(* CODESYS project l2sivacuum.library
   Company: SLAC
   Title: L2SI Vacuum Library
   Placeholder: L2SI Vacuum Library
   Version: 0.0.1

Project tree, tasks and I/O mapping:
  libraries: LCLS General, 0.1.4 (SLAC); Tc2_EtherCAT, * (Beckhoff Automation GmbH); Tc2_Standard, * (Beckhoff Automation GmbH); Tc2_System, * (Beckhoff Automation GmbH); Tc2_TcpIp, * (Beckhoff Automation GmbH); Tc2_Utilities, * (Beckhoff Automation GmbH); Tc3_Interfaces, * (Beckhoff Automation GmbH); Tc3_Module, * (Beckhoff Automation GmbH)
  DUTs/
    Gauges/
      data type E_PressureState
      data type Gauge_Type
      data type ST_VG
    Pumps/
      data type E_PumpState
      data type ST_AgilentPTM
      data type ST_EbaraDryPump
      data type ST_EbaraPTM
      data type ST_LeyboldPTM
      data type ST_PfeifferPTM
      data type ST_PIP
      data type ST_PTM
      data type ST_RoughPump
    Valves/
      data type E_ValvePositionState
      data type E_VCN
      data type E_VGC
      data type ST_VCC
      data type ST_VCC_NO
      data type ST_VCN
      data type ST_VGC
      data type ST_VRC
  GVLs/
    global variables Constants
    global variables Global_Variables
  POUs/
    Functions/
      Gauges/
        function block FB_925 [ST]: ACT_IO
        function block FB_972 [ST]: ACT_IO
        function block FB_GCM [ST]: ACT_IO
        function block FB_MKS_937A [ST]
        function block FB_MKS_937B [ST]
        function block FB_MKS275 [ST]: IO
        function block FB_MKS317 [ST]: IO
        function block FB_MKS422 [ST]: IO
        function block FB_MKS500 [ST]: IO
        function block FB_MKS500_EP [ST]: IO
        function block FB_MKS722 [ST]: ACT_IO
        function block FB_PressureState [ST]
      Pumps/
        function block FB_EbaraDryPump [ST]: ACT_IO
        function block FB_PIP_Gamma [ST]: ACT_SetGauge, IO
        function block FB_PTM_Agilent [ST]: BackingPressureSetPoint, ErrorMessage, IO
        function block FB_PTM_Ebara [ST]: ACT_IO, BackingPressureSetPoint
        function block FB_PTM_MagDriveDigital [ST]: ACT_IO
        function block FB_PTM_Pfeiffer [ST]
        function block FB_ScrollPump [ST]: IO
        function block FB_TurboExtLogic [LD]
      Valves/
        function F_TURBO_VRC_ILK [ST]
        function F_VALVE_REL_ILK [ST]
        function F_VRC_DIODE_ILK [ST]
        function block FB_TurbVentvalve_NO [LD]
        function block FB_VCC [ST]: ACT_IO
        function block FB_VCN [ST]: ACT_IO
        function block FB_VGC [ST]: ACT_IO, ACT_ResetAlarms
        function block FB_VRC [ST]: ACT_IO, F_TURBO_VRC_ILK
        function block FB_VRC_OK_CLS [ST]
  Version/
    global variables Global_Version
  VISUs/
*)

// DUTs/Gauges/E_PressureState
TYPE E_PressureState :
(
	//Valid States (Positive)
	Valid := gc_GaugeValidState, // gc_GaugeValidState set in "Global Variable Folder: Constants"
	ValidHi	:= 1, //gc_GaugeValidState + 1,
	ValidLo	:= 2, //gc_GaugeValidState + 2,
	
	// Invalid states
	PressInvalid	:= -1, //gc_GaugeValidState - 1,
	GaugeDisconnected	:=	-2, //gc_GaugeValidState -2,
	OoR	:= -6, //gc_GaugeValidState -6,
	// Ion gauges
	Off		:= -3, //gc_GaugeValidState - 3,
	Starting	:= -4 //gc_GaugeValidState - 4
) INT;
END_TYPE

// DUTs/Gauges/Gauge_Type
TYPE Gauge_Type: ( 
PG722B := 0, //Baraton Gauge
IG903 := 1 , //Cold Cathode
PG907 := 2 , //Pirani Gauge
IG909:= 3 , //Hot Cathode
PG925 := 4 ); //MicroPirani Gauge
(* This enumeration should match up with the EDM MUX button on the vacuum gauge expert controls screen *)
END_TYPE

// DUTs/Gauges/ST_VG
TYPE ST_VG :
STRUCT
	/// A general gauge structure is used to make the rest of the interlocking simpler. There are some parameters for cold cathodes that are not used by pirani.
	///These features aren't disabled, they just aren't used, think child/parent classes. 
	/// 
	{attribute 'pytmc' := '
    pv: PRESS
	io: i
    '}
	rPRESS: REAL;  //This is the human-readable pressure
	{attribute 'pytmc' := '
    pv: AT_VAC
	io: i
    '}
	xAT_VAC: BOOL;
	{attribute 'pytmc' := '
    pv: PRESS_OK
	io: i
    '}
	xPRESS_OK: BOOL;
	{attribute 'pytmc' := '
    pv: STATE
	io: i
    '}
	eState	:	E_PressureState;
	(* EPICS Controls *)	
	{attribute 'pytmc' := '
    pv: HV_SW
	io: io
    '}
	xHV_SW: BOOL; // High Voltage Switch from epics
	
	/// Controls and I/Os
	{attribute 'pytmc' := '
    pv: PRESS
	io: i
    '}
	i_iPRESS_R  :INT; // input Pressure // Link to analog Input
	{attribute 'pytmc' := '
    pv: HV_ON
	io: i
    '}
	i_xHV_ON	: BOOL; //  True when High Voltage is on  // 'TcLinkTo' (EL1124) ^Input
	{attribute 'pytmc' := '
    pv: DISC_ACTIVE
	io: i
    '}
	i_xDisc_Active : BOOL;// Discharge Current Active // 'TcLinkTo' (EL1124) ^Input
	{attribute 'pytmc' := '
    pv: HV_DIS
	io: i
    '}
	q_xHV_DIS : BOOL; // Enable High Voltage when True // 'TcLinkTo' (EL2624) ^Output
	//
	wHV_RO: WORD;
		
	/// Bakeout bit 
	xBAKEOUT: BOOL;
	
	//enum for gauge type - will replace iType
	eTYPE: Gauge_Type := PG907; 
	//Gauge type, deprecated (default to pirani)
	iTYPE: INT := 2;
	// Index location of the associated Pirani Gauge
	wPG: WORD;
	
	 
	xTurnOnTime: BOOL;/// Turn on Timers for cold cathode warmup
	iVacSp	:	INT;/// At vacuum setpoint for all gauges
	{attribute 'pytmc' := '
    pv: VAC_SP
	io:io
    '}
	rVAC_SP: REAL := 0.5;
	/// Protection setpoint for ion gauges at which the gauge turns off, not used for pirani 
	{attribute 'pytmc' := '
    pv: PRO_SP
	io: io
    '}
	rPRO_SP: REAL := 0.01;
	{attribute 'pytmc' := '
    pv: SP_HYS
	io: io
    '}
	/// Protection setpoint hysteresis 
	rHYS_PR: REAL; 
	/// Full scale pressure in Torr for baratron pressure conversion 
	rFULL_SCALE: REAL := 1000;
	
END_STRUCT
END_TYPE

// DUTs/Pumps/E_PumpState
TYPE E_PumpState :
(
pumpSTOPPED	:= 0,
pumpSTARTING	:= 1,
pumpRUNNING	:= 2,
pumpFAULT := 3

);
END_TYPE

// DUTs/Pumps/ST_AgilentPTM
TYPE ST_AgilentPTM EXTENDS ST_PTM :
STRUCT

(* Inputs *)
	(* 24V in Ramp state; 0V for others *)
	{attribute 'pytmc' := '
    pv: START
	io: i
	'}
    i_xSTART :	BOOL; 
	
	(* setpoint related to frequency *)
	{attribute 'pytmc' := '
    pv: R1Status
	io: i
	'}
	i_xR1	:  BOOL;
	
	(* setpoint related to Power *)
	{attribute 'pytmc' := '
    pv: R2Status
	io: i
	'}
	i_xR2	:  BOOL;
	
	(* low speed mode *)
	{attribute 'pytmc' := '
    pv: LSPD
	io: i
	'}
	i_xLSpd	:  BOOL;
	
	{attribute 'pytmc' := '
    pv: PUMP_CURRENT
	io: i
	'}
	i_iPumpCurrent: INT;
	(* Fault input*)
	//i_xFault : BOOL;  Inherit ST_PTM.xFault
	
	

(* controls *)
	(* Start/Stop - 
		q_RunDo ;   Inherit ST_PTM.
	 *)
	
	(* Low speed control *)
	{attribute 'pytmc' := '
    pv: LSPD_DO
	io: i
	'}
	q_xLSpd		:  BOOL; 
	
	(*Soft start *)
	{attribute 'pytmc' := '
    pv: XSS_DO
	io: i
	'}
	q_xSS   	:  BOOL; 
	
	(* Run interlock*)
	{attribute 'pytmc' := '
    pv: ILK_STATUS
	io: i
	'}
	xIlk : BOOL;
	
	{attribute 'pytmc' := '
    pv: STATE
	io: i
	'}	
	eState	:	E_PumpState;
	
	
	(*pump Lock*)
	{attribute 'pytmc' := '
    pv: FaultLock
	io: i
	'}
	xPumpFaultLock : BOOL := FALSE;
	// i_xPumpLockReset: BOOL := FALSE; Inherit ST_PTM.xReset
	// Error messages
	{attribute 'pytmc' := '
    pv: ErrorMessage
	io: i
	'}
	sError : STRING;

END_STRUCT
END_TYPE

// DUTs/Pumps/ST_EbaraDryPump
TYPE ST_EbaraDryPump EXTENDS ST_RoughPump :
STRUCT
(* Extension of the rough pump archetype for ebara 
Applicable to: 
EV-S20
EV-S50
EV-S100
EV-S200
*)

//Controls
{attribute 'pytmc' := '
    pv: MPStart
	io: i
    '}
q_xMPStart	:	BOOL; //Main Pump start
{attribute 'pytmc' := '
    pv: BPStart
	io: i
    '}
q_xBPStart	:	BOOL; // Booster Pump start (this can be started by the pump automatically)

xBPIlk	:	BOOL;	//Booster pump interlock
rBPIlkSP	:	REAL := 30; //Booster pump pressure setpoint
tonBP	:	TON := (PT:=T#5S); //Timer for pressure and valve stability


//Readbacks
{attribute 'pytmc' := '
    pv: MPStatus
	io: i
    '}
i_xMPStatus	:	BOOL; //MP status
{attribute 'pytmc' := '
    pv: BPStatus
	io: i
    '}
i_xBPStatus	:	BOOL; //BP status
{attribute 'pytmc' := '
    pv: WARN
	io: i
    '}
i_xWarning	:	BOOL; //Warning status
{attribute 'pytmc' := '
    pv: ALARM
	io: i
    '}
i_xAlarm	:	BOOL; //Alarm, maps to error
{attribute 'pytmc' := '
    pv: Remote
	io: i
    '}
i_xRemote	:	BOOL; //Remote control status


END_STRUCT
END_TYPE

// DUTs/Pumps/ST_EbaraPTM
TYPE ST_EbaraPTM EXTENDS ST_PTM :
STRUCT
(* Extension of the PTM archetype for Ebara turbo controllers 
Applicable to: 
ETC series
*)
//Controls
	{attribute 'pytmc' := '
    pv: START_SW
	io: io
	'}
i_xStart   : BOOL; //Momentary start switch
	{attribute 'pytmc' := '
    pv: STOP_SW
	io: io
	'}
i_xStop    : BOOL; //Momentary stop switch
// i_xReset is momentary reset switch - resets protection functions

	{attribute 'pytmc' := '
    pv: START
	io: i
	'}
q_xStart   : BOOL; //Outputs - FB decides if these are actually set
	{attribute 'pytmc' := '
    pv: STOP
	io: i
	'}
q_xStop    : BOOL;
	{attribute 'pytmc' := '
    pv: RESET
	io: i
	'}
q_xReset   : BOOL;
	{attribute 'pytmc' := '
    pv: ILK
	io: i
	'}
q_xProtection : BOOL; //NC. If opened, pump will decelerate/not start

iq_xSpeedSet    : BOOL; //Request to set speed
q_iSpeedSet   : DINT; //Requested speed (min. 100 RPM)

i_xOverride   : BOOL; //Override mode - ignores interlocks

//Readbacks - also has Accel/At speed/Decel/Fault/Cur Speed (min 100RPM)
	{attribute 'pytmc' := '
    pv: ROTATE_STATUS
	io: i
	'}
i_xRotate : BOOL; //If open, pump is rotating
	{attribute 'pytmc' := '
    pv: DECEL
	io: i
	'}
i_xDecel  : BOOL; //If closed, brake engaged (pump decelerating)
	{attribute 'pytmc' := '
    pv: FAULT_OK
	io: i
	'}
i_xNCFault  : BOOL; //Normally closed fault wiring. If false, there is a fault, or cable is unplugged.
	{attribute 'pytmc' := '
    pv: SPEED
	io: i
	'}
i_iRawSpeed	:	INT; //Raw pump speed from analog input

END_STRUCT
END_TYPE

// DUTs/Pumps/ST_LeyboldPTM
TYPE ST_LeyboldPTM EXTENDS ST_PTM :
STRUCT
(* Extension of the PTM archetype for Oerlikon turbo controllers 
Applicable to: 
Mag Drive Digital
Mag Drive S
More?
*)
//Readbacks
	{attribute 'pytmc' := '
    pv: DECEL
	io: i
	'}
	i_xDecel	:	BOOL;
	{attribute 'pytmc' := '
    pv: TEMP
	io: i
	'}
	i_diPumpTemp:	DINT;
	{attribute 'pytmc' := '
    pv: PWR
	io: i
	'}
	i_diPwr   	:   DINT;
	i_diElecTemp:	DINT;
	{attribute 'pytmc' := '
    pv: OVR_TEMP
	io: i
	'}
	i_xTempFault:	BOOL;
	i_xNCError	:	BOOL; //Using normally closed wiring

//Controls
	{attribute 'pytmc' := '
    pv: Remote_EN
	io: io
	'}
	q_xRemote : BOOL; (* Remote control enabled *)
END_STRUCT
END_TYPE

// DUTs/Pumps/ST_PfeifferPTM
TYPE ST_PfeifferPTM EXTENDS ST_PTM :
STRUCT
(* Extension of the PTM archetype for Pfeiffer turbos 
Applicable to: 
HiPace series w/ onboard controllers
More?
*)
//Readbacks
	i_diPwr		:	DINT;
	i_diElecTemp	:	DINT;
	i_diBtmTemp:	DINT;
	i_diBrngTemp:	DINT;
	i_diMtrTemp:	DINT;
	i_iErrorCode	:	INT; //might change these to enumeration someday
	i_iWarningCode	:	INT;
	i_xTempFault	:	BOOL;
	i_uiPowerPctRbk :   UINT;
	
//Controls
	q_uiPowerPct : UINT := 100; //Should normally be 100
	
END_STRUCT
END_TYPE

// DUTs/Pumps/ST_PIP
TYPE ST_PIP :
STRUCT
(* Read back *)
// 	i_xHVisON : BOOL; 
	
(* Interlock *)
	{attribute 'pytmc' := '
    pv: ExtIlk
	io: i
	'}
   	xHV_ExtIlk : BOOL; 
	{attribute 'pytmc' := '
    pv: ENB_SP
	io: io
	'}
	rHVEna_SP : REAL := 1.0E-4;	
	
(* EPICS Controls *)	
	{attribute 'pytmc' := '
    pv: HV_SW
	io: io
    '}
	xHVEna_SW : BOOL; 
	
(* IO Controls *)
	{attribute 'pytmc' := '
    pv: HV_DO
	io: i
    '}
	q_xHVEna_DO : BOOL;	// Enable High Voltage when True // 'TcLinkTo' (EL1124) ^Input
	{attribute 'pytmc' := '
    pv: PRESS
	io: i
    '}
	i_iPRESS: REAL;  //
	{attribute 'pytmc' := '
    pv: SP_DI
	io:i
    '}
	i_xSP_DI : BOOL; // NO contact // 'TcLinkTo' (EL1004) ^Input



END_STRUCT
END_TYPE

// DUTs/Pumps/ST_PTM
TYPE ST_PTM :
STRUCT
(* General PTM Structure
Each PTM might have a serial control structure, but all will have a general supervisory control structure

NOTE: This is an archetype, use an extension of this structure for a specific pump (or make one).

*)

(* Controls *)
	{attribute 'pytmc' := '
    pv: Run_SW
	io: io
	'}
	xRunSW	:	BOOL;
	{attribute 'pytmc' := '
    pv: Reset_SW
	io: io
	'}
	xReset	:	BOOL; //For resetting faults
	{attribute 'pytmc' := '
    pv: RUN_DO
	io: i
	'}
	q_RunDO 	:	BOOL;

(* Readbacks *)
{attribute 'pytmc' := '
    pv: RUN_OK
	io: i
	'}
	xExtRunOk	:	BOOL; (* also a control *)
	{attribute 'pytmc' := '
    pv: ACCEL
	io: i
	'}
	i_xAccel	:	BOOL;
	{attribute 'pytmc' := '
    pv: AT_SPD
	io: i
	'}
	i_xAtSpd	:	BOOL;
	i_diCurSpd	:	DINT;
	
	xCommTimeout	:	BOOL := TRUE;  (* Initialized true since we haven't talked to pump yet *)
(* Alarm Outputs *)
	{attribute 'pytmc' := '
    pv: FAULT
	io: i
	'}
	i_xFault		:	BOOL; //Note, for Ebara this is *false* in a fault condition!
	{attribute 'pytmc' := '
    pv: WARN
	io: i
	'}
	i_xWarn		:	BOOL; (* warning *)
	
(* IWS instructions *)
	xActive	:	BOOL; // this bit is set to add the pump to the system
	iPumpGrp 	:	INT; // all members of a pump group start at the same time
	
(* Operational Setpoints *)
	rForelineSP	:	REAL := 0.5;
	
	{attribute 'pytmc' := '
    pv: BackingPressureSP
	io: io
	'}
	rBackingPressureSP : REAL := 0.01;
	{attribute 'pytmc' := '
    pv: InletPressureSP
	io: io
	'}
	rInletPressureSP : REAL := 0.5;
	

END_STRUCT
END_TYPE

// DUTs/Pumps/ST_RoughPump
TYPE ST_RoughPump :
STRUCT
	
(* Generic roughing pump controls 

NOTE: This is an archetype, use an extension of this structure for a specific pump (or make one).

*)

//Controls
{attribute 'pytmc' := '
    pv: RUN_SW
	io: io
	'}
pv_xRunSW	:	BOOL; //epics/ software control switch
{attribute 'pytmc' := '
    pv: RUN_DO
	io: i
	'}
q_xRunDo 	:   BOOL; 

//Status and Readback
{attribute 'pytmc' := '
    pv: ILK_OK
	io: i
	'}
xIlk	:	BOOL; //Interlock bit, true means OK to run
xExtIlk	:	BOOL; //External interlock, this is where the logic goes
{attribute 'pytmc' := '
    pv: AT_SPD
	io: i
	'}
xAtSpd	:	BOOL; //Pump at speed setpoint
{attribute 'pytmc' := '
    pv: WARN
	io: i
	'}
xWrn	:	BOOL; //Pump warning
iWrn	:	BOOL; //Warning state/code
xErr	:	BOOL; //Error summary
iErr	:	BOOL; //Error state/code

END_STRUCT
END_TYPE

// DUTs/Valves/E_ValvePositionState
TYPE E_ValvePositionState :
	(
OPEN	:= 0,
CLOSED	:= 1,
MOVING	:= 2,
INVALID :=3
	);
END_TYPE

// DUTs/Valves/E_VCN
TYPE E_VCN :
	(
CloseValve	:= 0,
ControlValve	:= 1,
OpenValve	:= 2
	);
END_TYPE

// DUTs/Valves/E_VGC
TYPE E_VGC :
(

	Vented,
	AtVacuum,
	ERR_DiffPress,
	ERR_LostVac

);
END_TYPE

// DUTs/Valves/ST_VCC
TYPE ST_VCC :
STRUCT

(* Inputs *)
{attribute 'pytmc' := '
    pv: OPN_SW
	io: io
	'}
	pv_xOPN_SW	: BOOL;
	{attribute 'pytmc' := '
    pv:OVRD_OPN
	io: io
	'}
	xOvrdOpn	:	BOOL;
	{attribute 'pytmc' := '
    pv: OPN_OK
	io: i
	'}
	xOPN_OK	: BOOL;

(* Outputs *)
{attribute 'pytmc' := '
    pv: RUN_DO
	io: i
	'}
	q_xOPN_DO	: BOOL;

END_STRUCT
END_TYPE

// DUTs/Valves/ST_VCC_NO
TYPE ST_VCC_NO :
STRUCT

(* A normally open valve needs permission to close! *)
(* Inputs *)
{attribute 'pytmc' := '
    pv: CLS_SW
	io: io
	'}
	pv_xCLS_SW	: BOOL;
	{attribute 'pytmc' := '
    pv: OVRD_CLS
	io: io
	'}
	pv_xOvrdCls	:	BOOL;
	{attribute 'pytmc' := '
    pv: CLS_OK
	io: i
	'}
	xCLS_OK	: BOOL;

(* Outputs *)
{attribute 'pytmc' := '
    pv: CLS_DO
	io: i
	'}
	xCLS_DO	: BOOL;

END_STRUCT
END_TYPE

// DUTs/Valves/ST_VCN
TYPE ST_VCN :
STRUCT
	(* VCN - Valve Controlled Needle
	Used for Pfeiffer EVR 116 needle valves *)
	{attribute 'pytmc' := '
    pv: POS_RDBK
	io: i
    '}
	// Inputs
	i_iPosition	:	INT; //Position readback (if it exists)
	
	// Outputs
	{attribute 'pytmc' := '
    pv: POS_CTRL
	io: io
    '}
	q_iRawPosition	:	INT; //Position control 
	//For the EVR 116 this is 0-10V analog
	
	//Softvariables
	{attribute 'pytmc' := '
    pv: ILK_OK
	io: i
    '}
	xIlk	:	BOOL := FALSE; // Interlock Bit
	rUpperLimit	:	REAL;	//Upper limit on valve open
	rReqPosition	:	REAL; //Requested position (0.0-100.0%)
	eValveControl	:	E_VCN := CloseValve; // Valve control state

	ftIlk	:	F_TRIG;	

END_STRUCT
END_TYPE

// DUTs/Valves/ST_VGC
TYPE ST_VGC :
STRUCT

(* I/Os*)
(* Readbacks *)
	{attribute 'pytmc' := '
    pv: OPN_DI
	io: i
    '}
	i_xOpnLS	: BOOL;
	{attribute 'pytmc' := '
    pv: CLS_DI
	io: i
    '}
	i_xClsLS	: BOOL;
(* Controls *)
	{attribute 'pytmc' := '
    pv: OPN_DO
	io: i
    '}
	q_xOPN_DO	: BOOL;
	
	
(* EPICS Controls *)
	{attribute 'pytmc' := '
    pv: OPN_SW
	io: o
    '}
	pv_xOPN_SW	: BOOL;
	{attribute 'pytmc' := '
    pv: ALM_RST
	io: o
    '}
	pv_xAlmRst	: BOOL;
	{attribute 'pytmc' := '
    pv: OVRD_OPN
	io: o
    '}
	pv_xOvrdOpn	:	BOOL;

(* Interlocks *)
	{attribute 'pytmc' := '
    pv: DP_OK
	io: i
    '}
	xDP_OK	:	BOOL;	(* Managed by the VGC function (FB_VGC) *)// Indicates the valve can be opened because the differential pressure is low enough
	xEXT_OK	:	BOOL := FALSE;	(* External interlock for custom interlocking in addition to regular DP ilk, this must be set true, or the interlock condition before calling the FB_VGC *)
	{attribute 'pytmc' := '
    pv: OPN_OK
	io: i
    '}
	xOPN_OK	:	BOOL;	(* Final SUM of DP_OK and EXT_OK, needed because it allows the DP ilk to be switched off, see FB_VGC.Dis_DPIlk *)
	{attribute 'pytmc' := '
    pv: AT_VAC_SP
	io: o
    '}
	rAT_VAC_SP	:	REAL := 0.01;	// Interlock setpoint for gauges on both sides of valve
	rAT_VAC_SP_LAST	:	REAL :=0.01 ;	// Interlock setpoint for gauges on both sides of valve
	{attribute 'pytmc' := '
    pv: AT_VAC_HYS
	io: o
    '}
	rAT_VAC_HYS	:	REAL :=0.01;	// Hysteresis of the vacuum sp
	{attribute 'pytmc' := '
    pv: HYST_PERC
	io: o
    '}
	rHYST_PERC	:	REAL := 0.80;	// Hysteresis percentage
	{attribute 'pytmc' := '
    pv: AT_VAC
	io: i
    '}
	xAT_VAC	:	BOOL;	//At vacuum setpoint


(* Alarm Outputs *)
	xERR_DifPres		: 	BOOL;
	xERR_LstVac		: 	BOOL;
	xAlmSum			: 	BOOL;
	

	bErrorPresent : BOOL;
	iErrorCode: INT;
	sErrorMessage: STRING;

(*State*)	
	{attribute 'pytmc' := '
    pv: STATE
	io: i
    '}
	eVGC_State : E_VGC;
	{attribute 'pytmc' := '
    pv: POS_STATE
	io: i
    '}
	eState	:	E_ValvePositionState := INVALID;
	
END_STRUCT
END_TYPE

// DUTs/Valves/ST_VRC
TYPE ST_VRC :
STRUCT
(* Readbacks *)
	//If True, Valve is Open
	{attribute 'pytmc' := '
    pv: OPN_DI
	io: i
    '}
	i_xOpnLS	:	BOOL;
	//If True, Valve is Closed
	{attribute 'pytmc' := '
    pv: CLS_DI
	io: i
    '}
	i_xClsLS	:	BOOL;
	
	{attribute 'pytmc' := '
    pv: POS_STATE
	io: i
    '}
	eState	:	E_ValvePositionState := INVALID;

(* Inputs *)
	//Manually Pressing valve "Open/Close" on EDM
	{attribute 'pytmc' := '
    pv: OPN_SW
	io: io
    '}
	pv_xOPN_SW	: BOOL;
	//Manually toggling valve Local "ILK on button" on EDM
	{attribute 'pytmc' := '
    pv: OVRD_OPN
	io: io
    '}
	pv_xOvrdOpn	:	BOOL;
	//Calculated permissions to open valve
	{attribute 'pytmc' := '
    pv: OPN_OK
	io: i
    '}
	xOPN_OK	: BOOL;
	//In case VRC is normally open
	{attribute 'pytmc' := '
    pv: CLS_OK
	io: i
    '}
	xCLS_OK : BOOL := TRUE;
(* Outputs *)
	//When True, Opens valve
	//When False, Closes valve
	{attribute 'pytmc' := '
    pv: OPN_DO
	io: i
    '}
	q_xOPN_DO	: BOOL;

END_STRUCT
END_TYPE

// GVLs/Constants
VAR_GLOBAL CONSTANT
	gc_iSizeOfGGOArray : INT := 50;
	gc_GaugeValidState :	INT := 0;
END_VAR

// GVLs/Global_Variables
VAR_GLOBAL
	g_iSizeOfGGOArray : INT := 50;
	
	g_stSystem	:	System_Struct:= (
    	xFirstScan := TRUE
	);
	
	g_DummyVG	:	ST_VG;
	
	
	 fbGetCurTaskIdx : GETCURTASKINDEX;

END_VAR

// Version/Global_Version
{attribute 'TcGenerated'}
// This function has been automatically generated from the project information.
VAR_GLOBAL CONSTANT
	{attribute 'const_non_replaced'}
	{attribute 'linkalways'}
	stLibVersion_L2SI_Vacuum_Library : ST_LibVersion := (iMajor := 0, iMinor := 0, iBuild := 1, iRevision := 0, sVersion := '0.0.1');
END_VAR

// POUs/Functions/Gauges/FB_925
FUNCTION_BLOCK FB_925
VAR_INPUT
END_VAR
VAR_OUTPUT
	{attribute 'pytmc' := '
    pv: 
	'}
	PG	: ST_VG;
END_VAR
VAR_IN_OUT
	
END_VAR
VAR
	rV : REAL;
	fbGaugeState : FB_PressureState;
	rMaxPressure	:	REAL := 760; //Torr
	rMinPressure	:	REAL := 1E-5; //Torr
	
	(*IO*)
	i_iPRESS_R AT%I* :INT; // input Pressure // Link to analog Input
END_VAR

(* Standard MKS 9XX series conversion *)
(* works for 972 and 925 *)

//Default setpoint 50 mT
IF PG.rVAC_SP = 0 THEN
	PG.rVAC_SP := 5E-2;
END_IF

rV := 10*INT_TO_REAL(PG.i_iPRESS_R)/32767;

IF rV >= 0.99 THEN
	IF rV >= 0.99 AND rV < 1 THEN
		PG.rPRESS := 1E-5;
	ELSE
		PG.rPRESS := LREAL_TO_REAL(EXPT(10, rV-6));
	END_IF
	PG.xPRESS_OK := TRUE; //Backwards compatibility
ELSE
	PG.xPRESS_OK := FALSE;
END_IF

(* Pressure OK check *)
fbGaugeState.i_rV := rV;
fbGaugeState.i_MaxPressure := rMaxPressure;
fbGaugeState.i_MinPressure := rMinPressure;
fbGaugeState(iq_stVG:=PG);

(* Setpoint evaluation *)
PG.xAT_VAC := PG.xPRESS_OK AND (PG.rPRESS < PG.rVAC_SP);

ACTION ACT_IO:
PG.i_iPRESS_R :=i_iPRESS_R;
END_ACTION

END_FUNCTION_BLOCK

// POUs/Functions/Gauges/FB_PressureState
FUNCTION_BLOCK FB_PressureState
VAR_INPUT
	i_rV	:	REAL;
	i_rVMin	:	REAL := 0.01; // Anything less than this voltage is considered disconnected
	i_rVMax :	REAL := 10.5; // Anything more than this is considered invalid
	i_IGTurnOnTime	:	TIME := T#10S;
	
	i_MinPressure	:	REAL;
	i_MaxPressure	:	REAL;
END_VAR
VAR_OUTPUT
	q_eState 	:	E_PressureState;
END_VAR
VAR_IN_OUT
	iq_stVG	:	ST_VG;
END_VAR
VAR
	tonGaugeTurnOnTmr : TON;
END_VAR

(* Pressure State Evaluation
A. Wallace, 2016-8-31

This FB serves to evaluate the state of the pressure based on the raw voltage, pressure, and gauge state.

*)
// Is the gauge plugged in, and within a reasonable range?
IF i_rV < i_rVMin THEN
	q_eState := GaugeDisconnected;
ELSIF i_rV > i_rVMax THEN
	q_eState := PressInvalid;
ELSE
	// Is the gauge reading back a pressure that makes sense?
	CASE iq_stVG.eTYPE OF
		IG903:
			tonGaugeTurnOnTmr(IN:=iq_stVG.q_xHV_DIS, PT:=i_IGTurnOnTime, Q=>iq_stVG.xTurnOnTime);
			IF iq_stVG.q_xHV_DIS THEN
				IF tonGaugeTurnOnTmr.Q THEN
					IF iq_stVG.rPRESS >= i_MinPressure AND iq_stVG.rPRESS <= i_MaxPressure THEN
						q_eState := Valid;
					ELSE
						q_eState := OoR; 
					END_IF
				ELSE
						q_eState := Starting;
				END_IF
			ELSE
				q_eState := Off;
			END_IF
		IG909:
			IF iq_stVG.q_xHV_DIS THEN
				IF iq_stVG.rPRESS >= i_MinPressure AND iq_stVG.rPRESS <= i_MaxPressure THEN
					q_eState := Valid;
				ELSE
					q_eState := OoR;
				END_IF
			ELSE
				q_eState := Off;
			END_IF
		PG907, PG925, PG722B:
			IF iq_stVG.rPRESS >= i_MinPressure AND iq_stVG.rPRESS <= i_MaxPressure THEN
				q_eState := Valid;
			ELSIF iq_stVG.rPRESS < i_MinPressure THEN
				q_eState := ValidLo;
			ELSE
				q_eState := ValidHi;
			END_IF
		ELSE
			q_eState := PressInvalid;
	END_CASE
END_IF


iq_stVG.eState := q_eState;

// Legacy Press OK boolean eval
iq_stVG.xPRESS_OK := q_eState >= gc_GaugeValidState;

END_FUNCTION_BLOCK

// POUs/Functions/Gauges/FB_972
FUNCTION_BLOCK FB_972
VAR_INPUT
END_VAR
VAR_OUTPUT
	{attribute 'pytmc' := '
    pv: 
	'}
	VG	: ST_VG;
END_VAR
VAR_IN_OUT
	
END_VAR
VAR
	rV : REAL;
	(*IO*)
	i_iPRESS_R AT%I* :INT; // input Pressure // Link to analog Input
END_VAR

(* Standard MKS 9XX series conversion *)
(* works for 972 and 925 *)

rV := 10*INT_TO_REAL(VG.i_iPRESS_R)/32767;

IF rV > 1 THEN
	VG.rPRESS := LREAL_TO_REAL(EXPT(10, 2*rV-11));
	VG.xPRESS_OK := TRUE;
	VG.eState := Valid; //Press OK
ELSE
	VG.xPRESS_OK := FALSE;
	VG.eState := -6;
END_IF

ACTION ACT_IO:
VG.i_iPRESS_R :=i_iPRESS_R;
END_ACTION

END_FUNCTION_BLOCK

// POUs/Functions/Gauges/FB_GCM
FUNCTION_BLOCK FB_GCM
VAR_IN_OUT

END_VAR
VAR_OUTPUT
		{attribute 'pytmc' := '
    pv: 
	'}
	VG	:	ST_VG;
END_VAR
VAR
	rMinPressure: REAL;
	rV	:REAL;
	
	(*IO*)
	i_iPRESS_R AT%I* :INT; // input Pressure // Link to analog Input
END_VAR

(* Baratron Pressure Calc 
A. Wallace
2016-6-16
The full-scale pressure times the ratio of the meas.
voltage to full-scale voltage (10V).
The minimum pressure is always going to be 5e-4 * F.S.V.*)

rMinPressure := VG.rFULL_SCALE * 5E-4;


rV :=MAX((10*INT_TO_REAL(VG.i_iPRESS_R)/32767),0);
VG.rPRESS := (VG.rFULL_SCALE/10)*rV;
IF VG.rPRESS > rMinPressure THEN
	VG.xPRESS_OK := TRUE;
ELSE
	VG.xPRESS_OK := FALSE;
END_IF

(*IO soft linking*)
ACT_IO();

ACTION ACT_IO:
VG.i_iPRESS_R :=i_iPRESS_R;
END_ACTION

END_FUNCTION_BLOCK

// POUs/Functions/Gauges/FB_MKS_937A
FUNCTION_BLOCK FB_MKS_937A
VAR_IN_OUT
	VG : ST_VG;
END_VAR
VAR_INPUT
	PG	:	ST_VG := g_DummyVG;
END_VAR
VAR_OUTPUT
END_VAR
VAR
	rV	:	REAL;
END_VAR

(* 937A Logarithmic Output Conversion *)
(* 7-15-2015 *)
(* This function will read the pressure from any gauge on a 937A. *)

rV := 10*INT_TO_REAL(VG.i_iPRESS_R)/32767;
VG.rPRESS := LREAL_TO_REAL(EXPT(10,rV/0.6-12));


(* Ion Gauge Protection Functions *)
(* If the PG pressure is greater than the VG.PRO_SP then the gauge is disabled *)
(* If the PG pressure is less than the VG.PRO_SP then the gauge is enabled *)
(* This FB also implements some hysteresis so the gauge doesn't have rapid power cycling while near the turn on boundary *)

IF PG.rPRESS < VG.rPRO_SP THEN

VG.q_xHV_DIS := NOT VG.xHV_SW;

ELSIF NOT VG.q_xHV_DIS THEN
	IF VG.rPRESS > VG.rPRO_SP + VG.rHYS_PR OR PG.rPRESS > VG.rPRO_SP + VG.rHYS_PR THEN
		VG.q_xHV_DIS := TRUE;
	END_IF
ELSE
	VG.q_xHV_DIS := TRUE;
END_IF


(* Pressure gauge OK checks *)
VG.xPRESS_OK := (rV <=9.6 ) AND (rV>=0.6); //legacy

IF (rV <=9.6 ) AND (rV>=0.6) THEN
	VG.eState := Valid; // normal
ELSIF rV >= 0.18 AND rV <= 0.22 THEN
	VG.eState := ValidLo; //LO
ELSIF rV >= 9.7 AND rV<= 9.9 THEN
	VG.eState := ValidHi; //HIGH
ELSIF rV < 0.18 THEN
	VG.eState := GaugeDisconnected; //not on
ELSE
	VG.eState := PressInvalid; //other fault - could be no gauge, controller powering up etc
END_IF

(* Setpoint evaluation *)
VG.xAT_VAC := (VG.eState =Valid) AND VG.rPRESS < VG.rVAC_SP;

END_FUNCTION_BLOCK

// POUs/Functions/Gauges/FB_MKS_937B
FUNCTION_BLOCK FB_MKS_937B
VAR_IN_OUT
	
		PG	:	ST_VG := g_DummyVG;
END_VAR
VAR_INPUT
	
END_VAR
VAR_OUTPUT
	{attribute 'pytmc' := '
    pv: GCC
	'}
	VG : ST_VG;
	
	

END_VAR
VAR
	rV	:	REAL;
END_VAR

(* 937B Logarithmic Output Conversion *)
(* 5-20-2016, Alex Wallace and Scott Stubbs *)
(* This function will read the pressure from any gauge on a 937B. *)

rV := 10*INT_TO_REAL(VG.i_iPRESS_R)/32767;
VG.rPRESS := LREAL_TO_REAL(EXPT(10,(rV-7.2)/0.6));


(* Ion Gauge Protection Functions *)
(* If the PG pressure is greater than the VG.PRO_SP then the gauge is disabled *)
(* If the PG pressure is less than the VG.PRO_SP then the gauge is enabled *)
(* This FB also implements some hysteresis so the gauge doesn't have rapid power cycling while near the turn on boundary *)

IF PG.rPRESS < VG.rPRO_SP THEN

VG.q_xHV_DIS := NOT VG.xHV_SW;

ELSIF NOT VG.q_xHV_DIS THEN
	IF VG.rPRESS > VG.rPRO_SP + VG.rHYS_PR OR PG.rPRESS > VG.rPRO_SP + VG.rHYS_PR THEN
		VG.q_xHV_DIS := TRUE;
	END_IF
ELSE
	VG.q_xHV_DIS := TRUE;
END_IF


(* Pressure gauge OK checks *)
VG.xPRESS_OK := (rV <=9.6 ) AND (rV>=0.6);

IF (rV <=9.7 ) AND (rV>=0.6) THEN
	VG.eState := Valid; // normal
ELSIF rV >= 0.18 AND rV <= 0.22 THEN
	VG.eState := ValidLo; //LO
ELSIF rV > 9.7 AND rV<= 9.9 THEN
	VG.eState := ValidHi; //HIGH
ELSIF rV < 0.18 THEN
	VG.eState := GaugeDisconnected; //not on
ELSE
	VG.eState := PressInvalid; //other fault - could be no gauge, controller powering up etc
END_IF

(* Setpoint evaluation *)
VG.xAT_VAC := (VG.eState =Valid) AND VG.rPRESS < VG.rVAC_SP;

END_FUNCTION_BLOCK

// POUs/Functions/Gauges/FB_MKS275
FUNCTION_BLOCK FB_MKS275
VAR_IN_OUT

END_VAR
VAR_INPUT
END_VAR

VAR_OUTPUT
	{attribute 'pytmc' := '
    pv: 
	'}
	PG : ST_VG;
END_VAR
VAR
	MinPressure: REAL := 1E-4;
	V : REAL;
	Vlowest: REAL := 10;
	
	rValidLoBoundary	:	REAL := 0.375; // manual page 27
	rValidHiBoundary	:	REAL := 5.659;// 5.534; // manual page 27
	rDisconnectedBoundary	:	REAL := 0.3;
	
	(*IO*)
	i_iPRESS_R AT%I* :INT; // input Pressure // Link to analog Input
END_VAR

(* This function block is used to provide protection and automatic turn on of ion gauges,
 it also manages the turn on of the AT_VAC boolean, and checks to make sure the pressure is good *)
(* For MKS 275 mini-convectron *)

//Default setpoint 50 mT
IF PG.rVAC_SP = 0 THEN
	PG.rVAC_SP := 5E-2;
END_IF

(* Real-value calculation *)

V := 10*INT_TO_REAL(PG.i_iPRESS_R)/32767;	

Vlowest := MIN(V, Vlowest);

IF V > rDisconnectedBoundary AND V < rValidLoBoundary THEN

PG.rPRESS := MinPressure;
PG.eState := ValidLo;

ELSIF V >= rValidLoBoundary AND V < 2.842 THEN

PG.rPRESS := MAX( MinPressure, LREAL_TO_REAL( -0.02585 + 0.03767*V + 0.04563*EXPT(V,2)+ 0.1151*EXPT(V,3) - 0.04158*EXPT(V,4)+ 0.008737*EXPT(V,5)) );
PG.eState := Valid;

ELSIF V >= 2.842 AND V < 4.945 THEN

PG.rPRESS := LREAL_TO_REAL((0.1031-0.02322*V+0.07229*EXPT(V,2))/(1-0.3986*V+0.07438*EXPT(V,2)-0.006866*EXPT(V,3)));
PG.eState := Valid;

ELSIF V >= 4.945 AND V < rValidHiBoundary THEN

PG.rPRESS := LREAL_TO_REAL((100.624-20.5623*V)/(1-0.37679*V+0.0348656*EXPT(V,2)));
PG.eState := Valid;

ELSIF V <= rDisconnectedBoundary THEN

PG.eState := GaugeDisconnected; //Most likely not connected
PG.rPRESS := -1;;

ELSE
	
PG.eState := OoR; //Larger voltage, probably out of range?
PG.rPRESS := -1;
END_IF

(* Protection Functions *)
(* If the PG pressure is greater than the IG.PRO_SP then the gauge is disabled *)
(* If the PG pressure is less than the IG.PRO_SP then the gauge is enabled *)
(* This FB also implements some hysteresis so the gauge doesn't have rapid power cycling while near the turn on boundary *)

(* Pressure OK check *)
PG.xPRESS_OK := (PG.rPRESS >= MinPressure);

(* Setpoint evaluation *)
PG.xAT_VAC := PG.xPRESS_OK AND (PG.rPRESS<PG.rVAC_SP);

(*Soft IO Mapping *)
IO();

ACTION IO:
PG.i_iPRESS_R :=i_iPRESS_R;
END_ACTION

END_FUNCTION_BLOCK

// POUs/Functions/Gauges/FB_MKS317
FUNCTION_BLOCK FB_MKS317
VAR_IN_OUT
	
END_VAR
VAR_INPUT
	
END_VAR
VAR_OUTPUT
	{attribute 'pytmc' := '
    pv: 
	'}
	PG : ST_VG;
END_VAR
VAR
	rV	:	REAL;
		MinPressure: REAL := 1E-4;
		(*IO*)
	i_iPRESS_R AT%I* :INT; // input Pressure // Link to analog Input
END_VAR

(* 937B Logarithmic Output Conversion *)
(* 5-20-2016, Alex Wallace and Scott Stubbs *)
(* 09-28-2018, Margaret Ghaly *)
(* This function will read the pressure from any gauge on a 937B. *)

rV := 10*INT_TO_REAL(PG.i_iPRESS_R)/32767;
PG.rPRESS := LREAL_TO_REAL(EXPT(10,(rV-7.2)/0.6));


//Default setpoint 50 mT
IF PG.rVAC_SP = 0 THEN
	PG.rVAC_SP := 5E-2;
END_IF


(* Pressure gauge OK checks *)
PG.xPRESS_OK := (rV <=9.6 ) AND (rV>=0.6);

IF (rV <=9.7 ) AND (rV>=0.6) THEN
	PG.eState := Valid; // normal
ELSIF rV >= 0.18 AND rV <= 0.22 THEN
	PG.eState := ValidLo; //LO
ELSIF rV > 9.7 AND rV<= 9.9 THEN
	PG.eState := ValidHi; //HIGH
ELSIF rV < 0.18 THEN
	PG.eState := GaugeDisconnected; //not on
ELSE
	PG.eState := PressInvalid; //other fault - could be no gauge, controller powering up etc
END_IF

(* Pressure OK check *)
PG.xPRESS_OK := (PG.rPRESS >= MinPressure);

(* Setpoint evaluation *)
PG.xAT_VAC := (PG.eState =Valid) AND PG.rPRESS < PG.rVAC_SP;

ACTION IO:
PG.i_iPRESS_R :=i_iPRESS_R;
END_ACTION

END_FUNCTION_BLOCK

// POUs/Functions/Gauges/FB_MKS422
FUNCTION_BLOCK FB_MKS422
VAR_IN_OUT
		
END_VAR
VAR_INPUT
		PG	:	ST_VG;
END_VAR
VAR_OUTPUT
	{attribute 'pytmc' := '
    pv: GCC
	'}
	IG : ST_VG;
END_VAR
VAR
	rV	:	REAL;
	
	(*IOs to be linked*)
	/// Controls and I/Os
	i_iPRESS_R AT %I* :INT; // input Pressure // Link to analog Input
	q_xHV_DIS AT %Q* : BOOL; // Enable High Voltage when True // 'TcLinkTo' (EL2624) ^Output
	
	
END_VAR

(* 937B Logarithmic Output Conversion *)
(* 5-20-2016, Alex Wallace and Scott Stubbs *)
(* 09-28-2018, Margaret Ghaly *)
(* This function will read the pressure from any gauge on a 937B. *)

rV := 10*INT_TO_REAL(IG.i_iPRESS_R)/32767;
IG.rPRESS := LREAL_TO_REAL(EXPT(10,(rV-7.2)/0.6));



IF (rV <=9.7 ) AND (rV>=0.6) THEN
	IG.eState := Valid; // normal
ELSIF rV >= 0.18 AND rV <= 0.22 THEN
	IG.eState := ValidLo; //LO
ELSIF rV > 9.7 AND rV<= 9.9 THEN
	IG.eState := ValidHi; //HIGH
ELSIF rV < 0.18 THEN
	IG.eState := GaugeDisconnected; //not on
ELSE
	IG.eState := PressInvalid; //other fault - could be no gauge, controller powering up etc
END_IF


(* Ion Gauge Protection Functions *)
(* If the PG pressure is greater than the VG.PRO_SP then the gauge is disabled *)
(* If the PG pressure is less than the VG.PRO_SP then the gauge is enabled *)
(* This FB also implements some hysteresis so the gauge doesn't have rapid power cycling while near the turn on boundary *)

IF PG.rPRESS < IG.rPRO_SP THEN
	IG.q_xHV_DIS := IG.xHV_SW;

ELSIF IG.q_xHV_DIS THEN
	IF IG.rPRESS > (IG.rPRO_SP + IG.rHYS_PR) OR PG.rPRESS > (IG.rPRO_SP + IG.rHYS_PR) THEN
		IG.q_xHV_DIS := FALSE;
		IG.xHV_SW := FALSE;
	END_IF
ELSE
	IG.xHV_SW := FALSE;
END_IF

(* Pressure gauge OK checks *)
IG.xPRESS_OK := (rV <=9.6 ) AND (rV>=0.6);


(* Setpoint evaluation *)
IG.xAT_VAC := IG.xPRESS_OK AND IG.rPRESS < IG.rVAC_SP;


(*Soft IO Linking*)
// check ethercat Diagnostics
IO();

ACTION IO:
(*soft link inputs*)
IG.i_iPRESS_R:=	i_iPRESS_R; 

(*soft link outputs*)
q_xHV_DIS := IG.q_xHV_DIS;
END_ACTION

END_FUNCTION_BLOCK

// POUs/Functions/Gauges/FB_MKS500
FUNCTION_BLOCK FB_MKS500
VAR_IN_OUT

END_VAR
VAR_INPUT
	PG	:	ST_VG;
END_VAR
VAR_OUTPUT
	{attribute 'pytmc' := '
    pv: 
	'}
	IG : ST_VG;
END_VAR
VAR
	rV : REAL;
	pBase : REAL :=1.0E-10;//default curve base pressure is 1E-10. Confusing since can't actually read that low using analog out.
	vBase : REAL := 0; // corresponding vbase 0V based on default curve.  See manual pg. 44
	vSlope : REAL := 1.0; //looks correct for default curve
	GaugeTurnOnTmr : TON;
	MinPressure: REAL := 1E-10;
	cDefaultPressure : REAL := 0;
	
	
	(*IOs to be linked*)
	/// Controls and I/Os
	i_iPRESS_R AT %I* :INT; // input Pressure // Link to analog Input
	i_xHV_ON AT %I*	: BOOL; //  True when High Voltage is on  // 'TcLinkTo' (EL1124) ^Input
	i_xDisc_Active AT %I* : BOOL;// Discharge Current Active // 'TcLinkTo' (EL1124) ^Input
	q_xHV_DIS AT %Q* : BOOL; // Enable High Voltage when True // 'TcLinkTo' (EL2624) ^Output
	//
END_VAR

(* 500 Logarithmic Output Conversion, factory default configuration *)

rV := 10*INT_TO_REAL(IG.i_iPRESS_R)/32767;

(*
IF rV >= 0.49 AND rV < 0.52  THEN
	IG.wState := 5;
	IG.rPRESS := cDefaultPressure;
ELSIF rV < 0.4 THEN
	IG.wState := 4;//HV Off/ gauge disconnected
	IG.rPRESS := cDefaultPressure;
ELSE
	IG.wState := 1;
	IG.rPRESS := LREAL_TO_REAL(EXPT(10,((rV-vBase)/vSlope+LOG(pBase))));
END_IF
*)

(* Set Guage State based on the inputs HV ON and Discharge current*)
IF IG.i_xHV_ON AND NOT IG.i_xDisc_Active THEN
	IG.eState := Starting;
	IG.rPRESS := cDefaultPressure;
ELSIF IG.i_xHV_ON AND IG.i_xDisc_Active THEN
	IG.eState := Valid;
	IG.rPRESS := LREAL_TO_REAL(EXPT(10,((rV-vBase)/vSlope+LOG(pBase))));
ELSIF NOT IG.i_xHV_ON AND NOT IG.i_xDisc_Active THEN
	IG.eState := Off;
	IG.rPRESS := cDefaultPressure;
END_IF




(* Ion Gauge Protection Functions *)
(* If the PG pressure is greater than the VG.PRO_SP then the gauge is disabled *)
(* If the PG pressure is less than the VG.PRO_SP then the gauge is enabled *)
(* This FB also implements some hysteresis so the gauge doesn't have rapid power cycling while near the turn on boundary *)



IF PG.rPRESS < IG.rPRO_SP AND PG.xPRESS_OK THEN

	IG.q_xHV_DIS := IG.xHV_SW;

ELSIF IG.q_xHV_DIS THEN
	IF IG.rPRESS > (IG.rPRO_SP + IG.rHYS_PR)  OR PG.rPRESS > (IG.rPRO_SP + IG.rHYS_PR) THEN
		IG.q_xHV_DIS := FALSE;
		IG.xHV_SW := FALSE;
	END_IF
ELSE
	IG.q_xHV_DIS := FALSE;
	IG.xHV_SW := FALSE;
END_IF

(* Pressure gauge OK checks *)

GaugeTurnOnTmr(IN:=IG.q_xHV_DIS, PT:=T#10S, Q=>IG.xTurnOnTime);


//Backwards compatibility
IG.xPRESS_OK := (IG.eState = Valid) OR IG.xBAKEOUT;

(* Setpoint evaluation *)
IG.xAT_VAC := (IG.xPRESS_OK AND (IG.rPRESS < IG.rVAC_SP)) OR IG.xBAKEOUT AND (IG.eState = Valid) ;


(*Soft IO Linking*)
// check ethercat Diagnostics
IO();

ACTION IO:
(*check health of the ethercat terminal*) //todo
(*soft link inputs*)
IG.i_iPRESS_R:=	i_iPRESS_R; 
IG.i_xHV_ON:= i_xHV_ON;
IG.i_xDisc_Active:=i_xDisc_Active; 
(*soft link outputs*)
q_xHV_DIS := IG.q_xHV_DIS;
END_ACTION

END_FUNCTION_BLOCK

// POUs/Functions/Gauges/FB_MKS500_EP
FUNCTION_BLOCK FB_MKS500_EP
VAR_IN_OUT
		
END_VAR
VAR_INPUT

	PG	:	ST_VG;
END_VAR
VAR_OUTPUT
{attribute 'pytmc' := '
    pv: 
	'}
	IG : ST_VG;
END_VAR
VAR
	rV : REAL;
	pBase : REAL :=1.0E-10;//default curve base pressure is 1E-10. Confusing since can't actually read that low using analog out.
	vBase : REAL := 0; // corresponding vbase 0V based on default curve.  See manual pg. 44
	vSlope : REAL := 1.0; //looks correct for default curve
	GaugeTurnOnTmr : TON;
	MinPressure: REAL := 1E-10;
	cDefaultPressure : REAL := 0;
	
	
	(*IOs to be linked*)
	/// Controls and I/Os
	i_iPRESS_R AT %I* :INT; // input Pressure // Link to analog Input
	q_xHV_DIS AT %Q* : BOOL; // Enable High Voltage when True // 'TcLinkTo' (EP2624) ^Output
	//
END_VAR

(* 500 Logarithmic Output Conversion, factory default configuration *)


(*check health of the ethercat terminal*)

rV := 10*INT_TO_REAL(IG.i_iPRESS_R)/32767;

(* Set Guage State based on the inputs HV ON and Discharge current*)
IF rV >= 0.49 AND rV < 0.6  THEN
	IG.eState := Starting;
	IG.rPRESS := cDefaultPressure;
ELSIF rV < 0.4 THEN
	IG.eState := Off;
	IG.rPRESS := cDefaultPressure;
ELSE
	IG.eState := Valid;
	IG.rPRESS := LREAL_TO_REAL(EXPT(10,((rV-vBase)/vSlope+LOG(pBase))));
END_IF



(* Ion Gauge Protection Functions *)
(* If the PG pressure is greater than the VG.PRO_SP then the gauge is disabled *)
(* If the PG pressure is less than the VG.PRO_SP then the gauge is enabled *)
(* This FB also implements some hysteresis so the gauge doesn't have rapid power cycling while near the turn on boundary *)



IF PG.rPRESS < IG.rPRO_SP AND PG.xPRESS_OK THEN

	IG.q_xHV_DIS := IG.xHV_SW;

ELSIF IG.q_xHV_DIS THEN
	IF IG.rPRESS > (IG.rPRO_SP + IG.rHYS_PR)  OR PG.rPRESS > (IG.rPRO_SP + IG.rHYS_PR) THEN
		IG.q_xHV_DIS := FALSE;
		IG.xHV_SW := FALSE;
	END_IF
ELSE
	IG.q_xHV_DIS := FALSE;
	IG.xHV_SW := FALSE;
END_IF

(* Pressure gauge OK checks *)

GaugeTurnOnTmr(IN:=IG.q_xHV_DIS, PT:=T#10S, Q=>IG.xTurnOnTime);


//Backwards compatibility
IG.xPRESS_OK := (IG.eState = Valid) OR IG.xBAKEOUT;

(* Setpoint evaluation *)
IG.xAT_VAC := (IG.xPRESS_OK AND (IG.rPRESS < IG.rVAC_SP)) OR IG.xBAKEOUT AND (IG.eState = Valid) ;


(*Soft IO Linking*)
// check ethercat Diagnostics
IO();

ACTION IO:
(*soft link inputs*)
IG.i_iPRESS_R:=	i_iPRESS_R; 
(*soft link outputs*)
q_xHV_DIS := IG.q_xHV_DIS;
END_ACTION

END_FUNCTION_BLOCK

// POUs/Functions/Gauges/FB_MKS722
FUNCTION_BLOCK FB_MKS722
VAR_IN_OUT
	
END_VAR
VAR_OUTPUT
	{attribute 'pytmc' := '
    pv: 
	'}
	VG	:	ST_VG;
END_VAR
VAR_INPUT
	i_rMinPressure	:	REAL;
	i_rMaxPressure	:	REAL;
END_VAR
VAR
	rMinPressure: REAL;
	rVMin	:	REAL := 0.01; // Anything less than this voltage is considered disconnected
	rVMax :	REAL := 10.5; // Anything more than this is considered invalid
	rV	:REAL;
	
	(*IO*)
	i_iPRESS_R AT%I* :INT; // input Pressure // Link to analog Input
END_VAR


// Is the gauge plugged in, and within a reasonable range?
IF rV < rVMin THEN
	VG.eState := GaugeDisconnected;
ELSIF rV > rVMax THEN
	VG.eState := PressInvalid;
ELSIF VG.rPRESS >= rMinPressure AND VG.rPRESS <= i_rMaxPressure THEN
				VG.eState := Valid;
ELSIF VG.rPRESS < i_rMinPressure THEN
				VG.eState := ValidLo;
ELSE
				VG.eState := ValidHi;
END_IF
			
// Legacy Press OK boolean eval
VG.xPRESS_OK := VG.eState >= gc_GaugeValidState;

(*IO Soft Mapping*)
ACT_IO();

ACTION ACT_IO:
VG.i_iPRESS_R :=i_iPRESS_R;
END_ACTION

END_FUNCTION_BLOCK

// POUs/Functions/Pumps/FB_EbaraDryPump
FUNCTION_BLOCK FB_EbaraDryPump
VAR_INPUT
	i_stBPGauge	:	ST_VG; //booster pump interlock gauge
	i_xVlvOpn	:	BOOL; //valve(s) to main system load are open
END_VAR
VAR_OUTPUT
END_VAR
VAR_IN_OUT
	{attribute 'pytmc' := '
    pv: 
	'}
	stPump	:	ST_EbaraDryPump; //Ebara dry pump structure
END_VAR
VAR
	(*IO*)
	q_xMPStart	AT%Q*:	BOOL; //Main Pump start
	q_xBPStart	AT%Q*:	BOOL; // Booster Pump start (this can be started by the pump automatically)
	//Readbacks
	i_xMPStatus	AT%I*:	BOOL; //MP status
	i_xBPStatus	AT%I*:	BOOL; //BP status
	i_xWarning	AT%I*:	BOOL; //Warning status
	i_xAlarm	AT%I*:	BOOL; //Alarm, maps to error
	i_xRemote	AT%I*:	BOOL; //Remote control status
END_VAR

(* Ebara Dry Pump Control Routine
A. Wallace
2016-4-29
Applicable to:
EV-S20
EV-S50
EV-S100
EV-S200

Does basic controls for the pump. Starts booster pump when appropriate. Turns off pump
in the event of errors/ warnings. Provides interlocking interface.

Main Pump Operational Note:
Ebara recommends that the pump be exposed to the full system load after the main pump is running.

Booster Pump Operational Note:
The booster pump can either be started automatically by the pump itself (probably based on a timer?)
or it can be started by the PLC. The pressure setpoint is by default 30T. It may be wise to make
sure the pump was exposed to the full system load before starting the booster.

*)

//Mapping
ACT_IO();
// These are normally closed inputs
stPump.xErr := NOT stPump.i_xAlarm;
stPump.xWrn := NOT stPump.i_xWarning;


//Interlock and error/warning
stPump.xIlk :=  stPump.xExtIlk AND NOT (stpump.xErr OR stpump.xWrn);

//Start/ Stop the pump
IF stpump.xIlk THEN
	stpump.q_xMPStart := stpump.pv_xRunSW;
ELSE
	stpump.q_xMPStart := stpump.pv_xRunSW := FALSE;
END_IF

//Booster pump
stpump.xBPIlk := i_xVlvOpn AND stpump.i_xMPStatus AND (i_stBPGauge.rPRESS < stpump.rBPIlkSP) AND i_stbpgauge.xPRESS_OK;
stpump.tonBP(IN:=stpump.xBPIlk);
stpump.q_xBPStart := stpump.tonBP.Q;

ACTION ACT_IO:
(*Outputs*)
q_xMPStart	:= stPump.q_xMPStart;
q_xBPStart	:= stPump.q_xBPStart;
(*Inputs*)
stPump.i_xMPStatus:=	i_xMPStatus;
stPump.i_xBPStatus:=	i_xBPStatus;
stPump.i_xWarning:= i_xWarning	;
stPump.i_xAlarm:=	i_xAlarm;
stPump.i_xRemote:= i_xRemote;
END_ACTION

END_FUNCTION_BLOCK

// POUs/Functions/Pumps/FB_PIP_Gamma
FUNCTION_BLOCK FB_PIP_Gamma
VAR_INPUT
	i_stGauge	:	ST_VG; //Ion or Pirani gauge for pump interlock 
END_VAR
VAR_OUTPUT
	{attribute 'pytmc' := '
    pv: 
	'}
	stPump	:	ST_PIP; //Gamma Ion pump structure
	q_IG	:	ST_VG; //When ion pump is used as a measuring device for interlocking gate valves
END_VAR
VAR_IN_OUT
END_VAR
VAR
 rPRESS : REAL;
 rV : REAL;
 (* IO Controls *)
 q_xHVEna_DO AT %Q*: BOOL;	// Enable High Voltage when True // 'TcLinkTo' (EL1124) ^Input
 i_iPRESS  AT %I*: INT;  //
 i_xSP_DI  AT %I* : BOOL; // NO contact // 'TcLinkTo' (EL1004) ^Input

END_VAR

(* Does Gamma Ion pump HV interlock. Enable HV only when interlock gauge press is less than 1.0E-4 Torr *)

(* Interlock *)
IF (i_stGauge.xPRESS_OK AND (i_stGauge.rPRESS <= stPump.rHVEna_SP)) THEN
	stPump.xHV_ExtIlk := TRUE;
ELSE
	stPump.xHVEna_SW := FALSE;
	stPump.xHV_ExtIlk  := FALSE;
END_IF
(* Enable HV *)
stPump.q_xHVEna_DO := stPump.xHVEna_SW AND stPump.xHV_ExtIlk ;

(*Update output gauge values*)
ACT_SetGauge();
(*Soft IO Mapping*)
IO();

ACTION ACT_SetGauge:
(* convert the analog input into readable pressure*)
(* use logarithmic Pressure calculation, Output= Normal and Offset = 0*)
rV := 10*INT_TO_REAL(i_iPress)/32767;
rPRESS := LREAL_TO_REAL(EXPT(10,(rV-0))); (*offset = 0*)

IF (stPump.i_xSP_DI) THEN 
	q_IG.rPRESS := rPRESS;
	q_IG.xPRESS_OK := TRUE;
	ELSE
	q_IG.rPRESS := rPRESS;
	q_IG.xPRESS_OK := FALSE;
END_IF
END_ACTION

ACTION IO:

(*inputs*)
stPump.i_iPRESS:=	i_iPRESS;  
stPump.i_xSP_DI:=	i_xSP_DI;
(*output*)
q_xHVEna_DO:=stPump.q_xHVEna_DO;
END_ACTION

END_FUNCTION_BLOCK

// POUs/Functions/Pumps/FB_PTM_Agilent
FUNCTION_BLOCK FB_PTM_Agilent
VAR_IN_OUT
	{attribute 'pytmc' := '
    pv: 
	'}
	iq_stPtm	:	ST_AgilentPTM;	
END_VAR
VAR_INPUT
	i_stGauge	:	ST_VG; //Pirani backing gauge for pump interlock 
	i_rMaxBackingPressure : REAL;
END_VAR
VAR_OUTPUT
	
END_VAR
VAR
	//xRunOk	:	BOOL;
	nMaxR1Fault: INT :=5;
	nR1Fault : INT;
	tFaultWindowDuration : TIME := T#300S;
	tR1FaultDuration : TIME := T#120S;
	tTimeOutDuration: TIME:= T#120S;
	tFaultWindowElapsed: TON;
	tR1Fault : TON;
	tStartTimeOut : TON;
	tR1TimeOut: TON;
	step : INT :=0;
	nErrorCode: INT :=0;
	xBackingPressureOK: BOOL;
	
	
	(*I/Os*)
	i_xSTART 	AT%I*:	BOOL; // 'TcLinkTo' (EL1088) ^Input
	i_xR1	AT%I*	:  BOOL;// 'TcLinkTo' (EL1088) ^Input
	i_xR2	AT%I*	:  BOOL;// 'TcLinkTo' (EL1088) ^Input
	i_xLSpd	AT%I*:  BOOL;// 'TcLinkTo' (EL1088) ^Input
	i_iPumpCurrent AT%I*: INT;
	i_xFault AT%I*	:	BOOL;
	q_RunDO AT%Q*	:	BOOL;
	q_xLSpd	AT%Q*	:  BOOL;
	
END_VAR

(* Basic Agilent Turbo Controls *)
(* M. Ghaly, 2018-9-26 *)
(* state machine *)
CASE (step) OF
(*Pump Stopped State*)
	0: // Pump Stopped State
		iq_stPtm.xRunSW:=FALSE;
		//Reset Output signals;
		iq_stPtm.q_RunDO:=FALSE;
		iq_stPtm.q_xSS := FALSE;
		iq_stPtm.q_xLSpd:= FALSE;
		//Reset timer
		tFaultWindowElapsed.IN := FALSE;
		nR1Fault := 0;
		iq_stPtm.eState := pumpSTOPPED;
		step :=10;
(*Idle State waiting to start*)	
	10: // Idle State, waiting for the xRunSwitch
		IF iq_stPtm.xIlk  AND iq_stPTM.xRunSW THEN
			iq_stPtm.q_RunDO := iq_stPTM.xRunSW; //
			step:=20;
		END_IF
(*Pump Starting State*)	
	20: // Pump is starting
		nErrorCode:=0;
		iq_stPtm.q_RunDO := iq_stPTM.xRunSW; // done in previous state
		IF (*(NOT iq_stPtm.i_xR1) AND*)iq_stPtm.i_xSTART  THEN
		iq_stPtm.eState := pumpSTARTING;
		step:= 40;
		ELSIF tStartTimeOut.Q THEN
			step:=90; // or fault state
			nErrorCode:=950;
		END_IF
		// should check R1 ?? check Fault condition?
		
	40: // Pump is starting
		iq_stPtm.eState := pumpSTARTING;
		IF   NOT iq_stPtm.i_xR1 AND NOT iq_stPtm.i_xSTART  THEN
			step := 0 ;
		ELSIF NOT iq_stPtm.i_xR1 AND iq_stPtm.i_xSTART  THEN
			step :=40;
		ELSIF iq_stPtm.i_xR1 AND NOT iq_stPtm.i_xSTART THEN
			step:= 50;
		END_IF
		IF tR1TimeOut.Q THEN
			step:= 90;
			iq_stPtm.xPumpFaultLock := TRUE;
			nErrorCode:= 930; // R1 Signal at Start time out.
		END_IF
		
	50: // Pump is Running (Normal Operation) ( R1 is True and STARTing is FALSE)
		iq_stPtm.eState := pumpRUNNING;
		IF NOT iq_stPtm.i_xR1 THEN
			nR1Fault:= nR1Fault+1 ; 
			tFaultWindowElapsed.IN := TRUE; ///
			//tR1Fault.IN := TRUE;
			step :=60;
		END_IF
	
	60: // Pump is Running (Not Nomral Operation) (R1 is False, pump not @ speed )
		IF ((nR1Fault = nMaxR1Fault) AND NOT tFaultWindowElapsed.Q) OR (tR1Fault.Q) THEN // number of fault occured during the same time window
			step:= 90;
			tR1Fault.IN := FALSE;
			tFaultWindowElapsed.IN := FALSE;
			iq_stPtm.xPumpFaultLock := TRUE;
			nErrorCode:= 920; // R1 Signal Lost multiple times.
		ELSIF tFaultWindowElapsed.Q  THEN
			tFaultWindowElapsed.IN := FALSE;
			nR1Fault := 0;
		ELSIF iq_stPtm.i_xR1 THEN
			tR1Fault.IN := FALSE;
			step:=50;
		END_IF
	
	90: // Pump Fault STATE 
		iq_stPtm.xRunSW:=FALSE;
		iq_stPtm.q_RunDO:=FALSE;
		iq_stPtm.q_xSS := FALSE;
		iq_stPtm.q_xLSpd:= FALSE;
		iq_stPtm.eState := pumpFAULT;
		step := 95;
	
	95:	
		IF (NOT iq_stPtm.xPumpFaultLock) OR iq_stPtm.xRunSW THEN 
			step:=0;
		END_IF
END_CASE

(* Interrupts *)
(* FAULT signal*)
IF (iq_stPtm.i_xFault) AND (step < 90 ) THEN 
	iq_stPtm.eState := pumpFAULT; // no need taken care of in the state
	iq_stPtm.xPumpFaultLock := TRUE;
	nErrorCode := 900; // Pump Controller FAULT
	step:=90; 
END_IF


(*Pump Lock Reset bit*)
IF (iq_stPtm.xReset ) THEN
	iq_stPtm.xReset := FALSE;
	iq_stPtm.xPumpFaultLock := FALSE;
END_IF

(*Check backing gauge pressure*)
//xBackingPressureOK := i_stGauge.xPRESS_OK AND ( i_stGauge.rPRESS < iq_stPtm.rBackingPressureSP);

(* Interlock Sum *)
iq_stPtm.xIlk := iq_stPtm.xExtRunOk AND NOT iq_stPtm.i_xFault AND NOT iq_stPtm.xPumpFaultLock;// AND xBackingPressureOK;

IF NOT iq_stPtm.xIlk AND (NOT (step >= 90)) THEN
	step:=0; 
END_IF

(*Stop By the Operator and not due to fault *)
IF (NOT iq_stPtm.xRunSW) AND (NOT (step >= 90)) AND (NOT (step = 10)) THEN
	step := 0;
END_IF



(* Timers *)
tFaultWindowElapsed(PT:=tFaultWindowDuration);
tR1Fault(IN:= (step = 60), PT:=tR1FaultDuration);
tStartTimeOut(IN := (step=20), PT:=tTimeOutDuration);
tR1TimeOut(IN := (step=40), PT:=tTimeOutDuration);

IO();
(*Assign Error Message*)
iq_stPtm.sError := ErrorMessage(nErrorCode, iq_stPtm.eState);
(*Validate Backing Pressure set point doesn't exceed the Maximum backingPressure*)
iq_stPtm.rBackingPressureSP := BackingPressureSetPoint(iq_stPtm.rBackingPressureSP,i_rMaxBackingPressure);

METHOD BackingPressureSetPoint : REAL
VAR_INPUT
	i_SetPoint : REAL;
	rMaxBackingPressure: REAL;
END_VAR
BackingPressureSetPoint := Min(i_SetPoint , rMaxBackingPressure);
END_METHOD

METHOD PUBLIC ErrorMessage : STRING
VAR_INPUT
	nErrorCode : INT;
	eState: E_PumpState;
END_VAR
IF (eState := pumpFAULT ) THEN
	CASE nErrorCode OF
		950:
			ErrorMessage := 'Pump Starting Fault';
		930: 
			ErrorMessage := 'R1 Signal Timeout at Startup';
	
		920:
			ErrorMessage := 'R1 signal lost multiple times';

		900:
			ErrorMessage := 'Pump Controller Fault';	
	END_CASE
	
END_IF
END_METHOD

ACTION IO:
(*inputs*)
iq_stPtm.i_xSTART:=	i_xSTART;
iq_stPtm.i_xR1:=	i_xR1;
iq_stPtm.i_xR2:=	i_xR2;
iq_stPtm.i_xLSpd:=	i_xLSpd;
iq_stPtm.i_xFault:=	i_xFault;
(*outputs*)
q_RunDO := iq_stPtm.q_RunDO;
q_xLSpd := iq_stPtm.q_xLSpd;
i_iPumpCurrent := iq_stPtm.i_iPumpCurrent;
END_ACTION

END_FUNCTION_BLOCK

// POUs/Functions/Pumps/FB_PTM_Ebara
FUNCTION_BLOCK FB_PTM_Ebara
VAR_IN_OUT
	{attribute 'pytmc' := '
    pv: 
	'}
	iq_stPTM : ST_EbaraPTM;
END_VAR
VAR_INPUT
	i_iADCBits : UINT := 15;
	//i_iRawSpeed: INT; //Should come from PLC Soft IO.
	i_rMaxBackingPressure : REAL := 0.01;
	i_iMinSpeedRPM : INT := 100; //check pump manual for setting
	i_iMaxSpeedRPM : INT := 33600; // check pum manual for setting
END_VAR
VAR_OUTPUT

END_VAR
VAR
	TOF_START: TOF := (PT:=T#0.5S); //Manual states momentary switches need to be closed for >= 0.3s
	TOF_STOP: TOF := (PT:=T#0.5S);
	TOF_RESET: TOF :=(PT:=T#0.5S);
	
	TOF_SetSpeed: TOF :=(PT:=T#1S);
	
	(*IO*)
	(*inputs*)
	i_xDecel AT %I* : BOOL; //Link to brake input
	i_xAccel AT %I* : BOOL;
	i_xRotate AT %I* : BOOL;
	i_xNCFault AT %I* : BOOL;
	i_xAtSpeed AT %I* : BOOL;
	i_iRawSpeed AT %I* : INT; // Link to Analog input
	
	(*output*)
	q_xStart AT %Q* : BOOL; // link to output
	q_xStop AT %Q* : BOOL; //Link to output
	q_xReset AT %Q* : BOOL;
	q_xProtection AT %Q* : BOOL;
	q_xSetSpeed AT %Q* : BOOL;
	q_iSpeedSet AT %Q* :INT;	//Link to analog Output
	//more?
END_VAR

(* Ebara ETC control FB
Scott Stubbs & Alex W.
*)

(* Switch processing *)
TOF_START.IN := iq_stPTM.i_xStart;
TOF_START();
TOF_STOP.IN  := iq_stPTM.i_xStop;
TOF_STOP();
TOF_RESET.IN := iq_stPTM.xReset;
TOF_RESET();
///////////////////////
 (* to reset the Input speed OK bit *)
 TOF_SetSpeed (IN:= iq_stPTM.iq_xSpeedSet, Q => );
 IF NOT (TOF_SetSpeed.Q) THEN iq_stPTM.iq_xSpeedSet:= FALSE; 
 END_IF
 
//Normally closed fault handling
iq_stPTM.i_xFault := NOT iq_stPTM.i_xNCFault;

(* Simple protection reset *)
iq_stPTM.q_xProtection:= iq_stPTM.xExtRunOk;

(* Basic pump supervisory section *)
	(* If override mode, ignore everything else *)
IF iq_stPTM.i_xOverride THEN
	IF TOF_START.Q THEN
	iq_stPTM.q_RunDO:=TRUE;
	ELSIF TOF_STOP.Q THEN
		iq_stPTM.q_RunDO:=FALSE;
	END_IF
	//Handle faults - the way the Ebara cable is done, xFault is normally closed
ELSIF iq_stPTM.i_xFault OR (iq_stPTM.q_RunDO AND NOT iq_stPTM.xExtRunOk) THEN
	iq_stPTM.q_RunDO:=FALSE;
	iq_stPTM.q_xProtection:=FALSE;
	//And one for when we need to start the pump normally. Only allows pump to be started if ILK ok.
ELSIF TOF_START.Q AND iq_stPTM.xExtRunOk THEN
	iq_stPTM.q_RunDO:=TRUE;
	iq_stPTM.q_xStart:=TOF_START.Q;
//One section for when pump is told to stop
ELSIF TOF_STOP.Q THEN
		iq_stPTM.q_RunDO:=FALSE;
END_IF 

iq_stPTM.q_xReset:=TOF_RESET.Q; //No need for a conditional on these, code below takes care of it
iq_stPTM.q_xStop:=TOF_STOP.Q;
//Reset the start switch after processing
IF iq_stPTM.q_RunDO THEN
	iq_stPTM.q_xStart := TOF_START.Q;
END_IF

(* Pump speed calculation *)
IF iq_stPTM.i_iRawSpeed / (EXPT(2,i_iADCBits)-1) * 10 >= 0.2 THEN //Speed reading appears to zero at ~0.16V
iq_stPTM.i_diCurSpd := LREAL_TO_DINT(iq_stPTM.i_iRawSpeed/(EXPT(2,i_iADCBits)-1)*67000);
//V (AI/(2^{# ADC bits} -1 ) * 10[ADC 10V scaling]) * (33600 [Max RPM] - 100) / 5
ELSE
	iq_stPTM.i_diCurSpd := 0;
END_IF


(*Validate Backing Pressure set point doesn't exceed the Maximum backingPressure*)
iq_stPtm.rBackingPressureSP := BackingPressureSetPoint(iq_stPtm.rBackingPressureSP,i_rMaxBackingPressure);
(*soft IO mapping*)
ACT_IO();

ACTION ACT_IO:
(*soft io mapping*)
(*inputs*)

iq_stPTM.i_xDecel := i_xDecel ;
iq_stPTM.i_xAccel :=	i_xAccel ;
iq_stPTM.i_xRotate :=	i_xRotate;
iq_stPTM.i_xNCFault :=	i_xNCFault ;
//iq_stPTM.i_xAtSpeed := i_xAtSpeed;
iq_stPTM.i_iRawSpeed :=	i_iRawSpeed;
//V (AI/32767*10) * (33600 {Max RPM} - 100) / 5
(*outputs*)
q_xStart:= iq_stPTM.q_xStart;
q_xStop := iq_stPTM.q_xStop;
q_xReset := iq_stPTM.q_xReset;
q_xProtection := iq_stPTM.q_xProtection;
q_xSetSpeed := iq_stPTM.iq_xSpeedSet;
(*Validate Set Speed within range *) 
IF iq_stPTM.q_iSpeedSet  >= i_iMinSpeedRPM AND iq_stPTM.q_iSpeedSet  <=i_iMaxSpeedRPM THEN 
	q_iSpeedSet  := LIMIT(0, DINT_TO_INT((iq_stPTM.q_iSpeedSet - i_iMinSpeedRPM) / i_iMaxSpeedRPM *16383/5),16383); //Max 5V
	//:= DINT_TO_INT((q_iSpeedSet-100) / 33600 *32767/2); //Max 5V
END_IF
END_ACTION

METHOD PUBLIC BackingPressureSetPoint : REAL
VAR_INPUT
	i_SetPoint : REAL;
	rMaxBackingPressure: REAL;
END_VAR
BackingPressureSetPoint := Min(i_SetPoint , rMaxBackingPressure);
END_METHOD

END_FUNCTION_BLOCK

// POUs/Functions/Pumps/FB_PTM_MagDriveDigital
FUNCTION_BLOCK FB_PTM_MagDriveDigital
VAR_IN_OUT
	{attribute 'pytmc' := '
    pv: 
	'}
	iq_stPtm	:	ST_LeyboldPTM;
END_VAR
VAR_INPUT
END_VAR
VAR_OUTPUT

END_VAR
VAR
	xRunOk	:	BOOL;
	tofRemoteDelay	:	TOF;
	
	
	(*IO*)
	i_xAtSpd AT%I*: BOOL;
	i_xFault AT%I*: BOOL;
    i_xAccel AT%I*: BOOL;
 	i_xDecel AT%I*: BOOL;
 	i_xWarn AT%I*: BOOL;
	
	q_RunDO AT%Q*: BOOL;
	q_xRemote AT%Q*: BOOL;
END_VAR

(* Basic MagDrive Digital Turbo Controls *)
(* A. Wallace, 2015-7-15 *)

tofRemoteDelay(IN:=iq_stPtm.q_RunDO, PT:=T#5S);

iq_stPtm.q_xRemote := tofRemoteDelay.Q;

(* Interlock Sum *)
xRunOk := iq_stPtm.xExtRunOk AND NOT iq_stPtm.i_xFault;

(* Basic pump supervisory section *)
IF xRunOk THEN
	iq_stPtm.q_RunDO := iq_stPTM.xRunSW;
ELSE
	iq_stPtm.xRunSW:=FALSE;
	iq_stPtm.q_RunDO:=FALSE;
END_IF

(*I/O soft mapping*)
ACT_IO();

ACTION ACT_IO:
(*Inputs*)
iq_stPtm.i_xAtSpd := i_xAtSpd;
iq_stPtm.i_xFault := NOT i_xFault;
iq_stPtm.i_xAccel := i_xAccel;
iq_stPtm.i_xDecel := i_xDecel;
iq_stPtm.i_xWarn := i_xWarn;

(*Outputs*)
q_RunDO := iq_stPtm.q_RunDO;
q_xRemote := iq_stPtm.q_xRemote; // remote out
END_ACTION

END_FUNCTION_BLOCK

// POUs/Functions/Pumps/FB_PTM_Pfeiffer
FUNCTION_BLOCK FB_PTM_Pfeiffer
VAR_IN_OUT
	{attribute 'pytmc' := '
    pv: 
	'}
	iq_stPTM : ST_PfeifferPTM;
END_VAR
VAR_INPUT
END_VAR
VAR_OUTPUT
END_VAR
VAR
END_VAR

(* Basic pump supervisory section *)
IF iq_stPTM.xExtRunOk AND NOT (iq_stPTM.i_xFault OR iq_stPTM.i_xTempFault) THEN
	iq_stPTM.q_RunDO:=iq_stPTM.xRunSW;
ELSE
	iq_stPTM.xRunSW:=0;
	iq_stPTM.q_RunDO:=FALSE;
END_IF

END_FUNCTION_BLOCK

// POUs/Functions/Pumps/FB_ScrollPump
FUNCTION_BLOCK FB_ScrollPump
VAR_IN_OUT

END_VAR
VAR_OUTPUT
	{attribute 'pytmc' := '
    pv:
	'}
	iq_stPFO	:	ST_RoughPump;
END_VAR
VAR_INPUT
	TurboIsON : BOOL;
	VentValve	: ST_VCC_NO; // type of vent valve might change
END_VAR
VAR
	Tmr_TOF : TOF;
	tTimerDuration : Time:= T#150S;
	//Previous_RunSW : BOOL;
	// Digital Output to be linked
	q_xRunDo AT%Q*	:   BOOL; 
END_VAR

//Turn on scroll pump if the Turbo Vent Valve is closed. So you are not just
// pumping air and accomplishing nothing

// cannot turn off scroll pump if turb is running. delay scroll off 150s.  


Tmr_TOF(IN:=TurboIsON, PT := tTimerDuration);

IF VentValve.xCLS_DO THEN
	iq_stPFO.q_xRunDo := (Tmr_TOF.Q OR iq_stPFO.pv_xRunSW);
ELSE
	iq_stPFO.q_xRunDo := FALSE;
END_IF

iq_stPFO.pv_xRunSW := iq_stPFO.q_xRunDo;

iq_stPFO.pv_xRunSW := iq_stPFO.q_xRunDo;

(*soft io Mapping*)
IO();

ACTION IO:
q_xRunDo:= iq_stPFO.q_xRunDo;
END_ACTION

END_FUNCTION_BLOCK

// POUs/Functions/Pumps/FB_TurboExtLogic
FUNCTION_BLOCK FB_TurboExtLogic
VAR_IN_OUT
	Turbo		:	ST_AgilentPTM;
END_VAR
VAR_INPUT
	BackingGauge:	ST_VG;
	InletGauge	:	ST_VG;
	VentValve	:	ST_VCC_NO;
	ScrollPump	:	ST_RoughPump;
END_VAR
VAR_OUTPUT
END_VAR
VAR
END_VAR

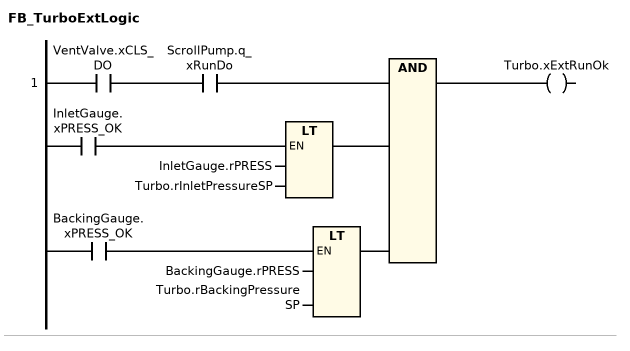
// NETWORK 1
Turbo.xExtRunOk := (VentValve.xCLS_DO AND ScrollPump.q_xRunDo) AND (InletGauge.xPRESS_OK AND InletGauge.rPRESS < Turbo.rInletPressureSP) AND (BackingGauge.xPRESS_OK AND BackingGauge.rPRESS < Turbo.rBackingPressureSP);

END_FUNCTION_BLOCK

// POUs/Functions/Valves/F_TURBO_VRC_ILK
FUNCTION F_TURBO_VRC_ILK : BOOL
VAR_INPUT

	i_xHiVac 	: BOOL;
	i_xRunPTM	: BOOL;
	i_xFLVac	: BOOL;

END_VAR
VAR

	rHysterisis : REAL := 0;

	xInterlock: BOOL;
	rTolerance: REAL := 20;
END_VAR

(* Close the vic if the roughing pump pirani loses its at-vac setpoint while the turbo is pumping *)
F_TURBO_VRC_ILK := (NOT i_xHiVac AND NOT i_xRunPTM AND NOT i_xFLVac) OR
					(NOT i_xRunPTM AND i_xFLVac) OR
					(i_xRunPTM AND i_xFLVac);

END_FUNCTION

// POUs/Functions/Valves/F_VALVE_REL_ILK
FUNCTION F_VALVE_REL_ILK : BOOL
VAR_INPUT
	i_stUSG	:	ST_VG;
	i_stDSG	:	ST_VG;
	//Orders of magnitude allowed between up/downstream pressures for valve to open. Must be real positive integer.
	i_iOrdersMagnitude: INT;
END_VAR
VAR
	rPressRatio : REAL;
	rMaxRatioAllowed	:	LREAL := EXPT(10,i_iOrdersMagnitude);
	rMinRatioAllowed	:	LREAL := EXPT(10,(-i_iOrdersMagnitude));
END_VAR

(* S. Stubbs 11/2015 *)

(* OK, this is going to be a general-use function that will return whether the ratio of the pressures given is less than x orders of magnitude.
True iff 10^(-x) < a/b < 10^x.  Simple, right?  Just make sure it gets a positive order of magnitude and the pressures aren't 0. ~Scott *)   

(* Find ratio *)

IF i_stDSG.rPRESS <> 0 THEN
	rPressRatio := i_stUSG.rPRESS / i_stDSG.rPRESS;

	F_VALVE_REL_ILK := rPressRatio < rMaxRatioAllowed AND rMinRatioAllowed < rPressRatio;
ELSE
	F_VALVE_REL_ILK := FALSE;
END_IF

END_FUNCTION

// POUs/Functions/Valves/F_VRC_DIODE_ILK
FUNCTION F_VRC_DIODE_ILK : BOOL
VAR_INPUT

	i_stPGA : ST_VG;
	i_stPGB	: ST_VG;

END_VAR
VAR

	rHysterisis : REAL := 0;

	xInterlock: BOOL;
	rTolerance: REAL := 20;
END_VAR

(* The principle is simple, a VRC should never open when B side pressure is greater than the A side pressure. *)
rTolerance := 20;
F_VRC_DIODE_ILK := ((i_stPGA.rPRESS + rTolerance >= i_stPGB.rPRESS + rHysterisis) OR i_stPGA.xBAKEOUT) AND i_stPGA.xPRESS_OK AND i_stPGB.xPRESS_OK;

(* OK it gets a bit more complicated with hysterisis,

Now, if the F_VIC_DIODE_ILK is FALSE then some hysterisis is added to the B side. But if it's OK then we just stick with making sure that the A side is greater than the B side

*)
(*
IF NOT F_VIC_DIODE_ILK THEN
Hysterisis := 40;
ELSE
Hysterisis := 0;
END_IF
*)

END_FUNCTION

// POUs/Functions/Valves/FB_TurbVentvalve_NO
FUNCTION_BLOCK FB_TurbVentvalve_NO
VAR_IN_OUT
	iq_stValve : ST_VCC_NO;
END_VAR
VAR_INPUT
	i_stPTM	: ST_AgilentPTM;
END_VAR
VAR
	tofTmr 		: 	TOF;
END_VAR

(*If the turbo is on, you cannot open the valve. In order to open the valve, you have to allow the turbopump
 to have already been turned off for 2 minutes and you have to press the open button on the vent valve

If the code looks confusing please use a truth table to verify*)

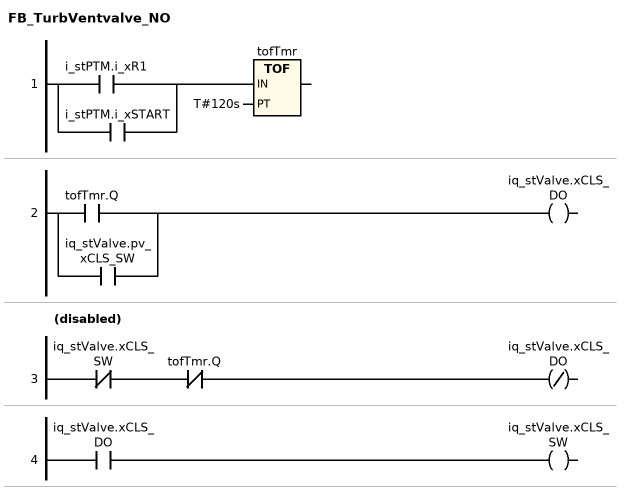
// NETWORK 1
tofTmr(IN := i_stPTM.i_xR1 OR i_stPTM.i_xSTART, PT := T#120s); // TOF

// NETWORK 2
iq_stValve.xCLS_DO := tofTmr.Q OR iq_stValve.pv_xCLS_SW;

// NETWORK 3 (disabled)
// iq_stValve.xCLS_DO := NOT (NOT iq_stValve.xCLS_SW AND NOT tofTmr.Q);

// NETWORK 4
iq_stValve.xCLS_SW := iq_stValve.xCLS_DO;

END_FUNCTION_BLOCK

// POUs/Functions/Valves/FB_VCC
FUNCTION_BLOCK FB_VCC
VAR_IN_OUT

END_VAR
VAR_INPUT

END_VAR
VAR_OUTPUT
	{attribute 'pytmc' := '
    pv:
	'}
	iq_stValve : ST_VCC;
END_VAR
VAR

	tonOvrd	:	TON;
	tonDelOK : TON;
	rtOK	:	R_TRIG;

	(*IO*)
	q_xOPN_DO	AT%Q*: BOOL;

END_VAR


IF NOT iq_stValve.xOPN_OK THEN
iq_stValve.pv_xOPN_SW := FALSE;
END_IF

(* Override logic *)
(* Goal: give ability to override, but do so in a way that people won't forget it.
Solution: Override only after ten seconds of override, protect against blips,
when the valve permission goes true for more than ten seconds consistently, remove override
*)

tonDelOK(IN:=iq_stValve.xOPN_OK, PT:=T#10S);
rtOK(CLK:=tonDelOK.Q);
IF rtOK.Q THEN iq_stValve.xOvrdOpn :=FALSE; END_IF

//Override timer
tonOvrd(IN:=iq_stValve.xOvrdOpn, PT:=T#10S);

(* Here's where the valve opens *)
iq_stValve.q_xOPN_DO := (iq_stValve.pv_xOPN_SW AND iq_stValve.xOPN_OK) OR (tonOvrd.Q AND g_stSystem.xOverrideMode);

(*IO Mapping*)
ACT_IO();

ACTION ACT_IO:
(*outputs*)
q_xOPN_DO:= iq_stValve.q_xOPN_DO;
END_ACTION

END_FUNCTION_BLOCK

// POUs/Functions/Valves/FB_VCN
FUNCTION_BLOCK FB_VCN
VAR_INPUT
	i_xExtIlk	:	BOOL; //External Interlock
	i_ReqPos	:	BOOL; //Requested position
END_VAR
VAR_OUTPUT
	{attribute 'pytmc' := '
    pv:
	'}
	iq_stVCN	:	ST_VCN; //Needle valve structure
END_VAR
VAR_IN_OUT
	
END_VAR

VAR CONSTANT
	rOpenVoltage	:	REAL := 9.1; // From the EVR 116 manual
	rCloseVoltage	:	REAL := 0.4;	
END_VAR
VAR
	// Requested voltage
	rReqVoltage: REAL := 0;
	(*IO*)
	q_iRawPosition AT%Q* :INT;
END_VAR

(* Needle valve control FB
A. Wallace 2016-7-21

This FB should be used as a low level control block.

It provides:

Valve position ceiling
Interlock
Scaling

It is not intended for:
Closed-loop control

It could be used for:
Valve position/flow linearization

Note: Raw position calc is based on 0.5 to 9V span, 32767 bits
*)




// Interlocking
iq_stVCN.xIlk := i_xExtIlk;

IF iq_stVCN.xIlk THEN
	
	IF iq_stVCN.eValveControl = OpenValve THEN
		iq_stVCN.rReqPosition := iq_stVCN.rUpperLimit;
	ELSIF iq_stVCN.eValveControl = CloseValve THEN
		iq_stVCN.rReqPosition := 0;
	ELSE
		 ;
	END_IF

	//Raw position calc
	iq_stVCN.rReqPosition := LIMIT(0, iq_stVCN.rReqPosition, iq_stVCN.rUpperLimit);
	rReqVoltage := iq_stVCN.rReqPosition * (rOpenVoltage-rCloseVoltage)/100 + rCloseVoltage;
	rReqVoltage := LIMIT(rCloseVoltage, rReqVoltage, rOpenVoltage); //The requested voltage should remain within this range
	iq_stvcn.q_iRawPosition := REAL_TO_INT( 32767/10 * rReqVoltage);	
ELSE
	iq_stvcn.q_iRawPosition := 0;
	iq_stVCN.rReqPosition := 0;
	iq_stVCN.eValveControl := CloseValve;
END_IF

ACTION ACT_IO:
(*outputs*)
q_iRawPosition := iq_stVCN.q_iRawPosition;
END_ACTION

END_FUNCTION_BLOCK

// POUs/Functions/Valves/FB_VGC
FUNCTION_BLOCK FB_VGC
VAR_IN_OUT
	
END_VAR
VAR_INPUT
	(*Upstream Gauge, usually ion gauge*)
	i_stUSG	:	ST_VG;
	(*Upstream Gauge, usually ion gauge*)
	i_stDSG	:	ST_VG;
	{attribute 'pytmc' := '
    pv: Dis_DPIlk
	'}
	i_xDis_DPIlk : BOOL := FALSE;  (* Set to true when calling the function to disable the differential pressure interlock *)
	{attribute 'pytmc' := '
    pv: EPS_OK
	'}
	i_xEPS_OK:	BOOL	:= TRUE; (*External EPS interlock, Set to TRUE when no EPS interlock is required, otherwise set to correct interlock signal*)
	{attribute 'pytmc' := '
    pv: MPS_OK
	'}
	i_xPMPS_OK:	BOOL	; (*External MPS interlock, Set to TRUE when no PMPS interlock is required*)
	i_xExt_OK: BOOL; (*Other External Interlock*)
END_VAR
VAR_OUTPUT
	{attribute 'pytmc' := '
    pv:
	'}
	iq_stValve : ST_VGC; (* All valve data and states will be in this struct*)
	
	{attribute 'pytmc' := '
    pv: MPS_FAULT
	'}
	xMPS_FAULT:	BOOL; (*MPS Fast Fault, is set when the Valve is closed*)
END_VAR
VAR
	
	rDiffPressAllowed	:	REAL := 22.5; // Torr, Default value comes from Vat Valve Manual
	rDiffPress : REAL;
	set : BOOL;
    reset: BOOL;
	  
	xFirstPass	:	BOOL;
	fbFSInit		:	R_TRIG;
	
	tonDelOK : TON;
	rtOK	:	R_TRIG;
	tonOvrd	:	TON;
	
	tDelOK	:	TIME := T#10S;
	tOvrd	:	TIME := T#10s;
	
	
	(* Timeouts*)
	tTimeOutDuration: TIME:= T#180S;
	tOPNtimeout: TON;
	tCLStimeout:TON;
	
	
	(*IO*)
	i_xOpnLS	AT%I*: BOOL;
	i_xClsLS	AT%I*: BOOL;
	q_xOPN_DO	AT%Q*: BOOL;
	
END_VAR

(* Vacuum gate valve
A. Wallace
16-10-29

A gate valve isolates vacuum volumes. Ideally it can be opened when a system is vented
to allow for faster pumping, and will close when high vacuum is lost.

The following behavior is good for valves in something like a gas attenuator.
This function block does the following:
1. The valve can be opened when the difference between the pressures on both sides is
less than the maximum differential pressure.
2. This rule persists until the pressures on both sides are lower than the vacuum-setpoint.
3. Once at-vac, the valve will close if the pressure on either side rises above the setpoint.

Alternatively, the differential pressure interlock can be disabled so the valve may only be opened
if the pressure on both sides is lower than the at-vacuum-setpoint. You want this behavior if 
the valve is to be used in a UHV section.

Hysteresis is employed to ensure a smooth transition from vented/pumping down, to at-vac.

Finally, an override system is built in so you can bypass all the interlocking logic and 
get back online.
*)
(* 10/1/2018 Margaret Ghaly *)


fbFSInit( CLK := TRUE, Q => xFirstPass);

(* On first PLC pass, put valve into vented state, which implies a closed valve *)
IF xFirstPass THEN
	iq_stValve.eVGC_State := Vented;
	iq_stValve.pv_xOPN_SW := FALSE;
END_IF


///Check valve postion
IF iq_stValve.i_xClsLS AND  iq_stValve.i_xOpnLS THEN
	iq_stValve.eState:=INVALID;
ELSIF NOT iq_stValve.i_xClsLS AND iq_stValve.i_xOpnLS THEN 
	iq_stValve.eState:=OPEN;
ELSIF iq_stValve.i_xClsLS AND NOT iq_stValve.i_xOpnLS THEN 
	iq_stValve.eState:=CLOSED;
ELSIF NOT iq_stValve.i_xClsLS AND NOT iq_stValve.i_xOpnLS THEN 
	iq_stValve.eState:=MOVING;
ELSE
	iq_stValve.eState:=INVALID;
END_IF

// Update hysteresis
///////////////////////////////////////////////////
IF iq_stValve.rAT_VAC_SP_LAST <> iq_stValve.rAT_VAC_SP OR xFirstPass THEN
	iq_stValve.rAT_VAC_SP_LAST := iq_stValve.rAT_VAC_SP;
	iq_stValve.rAT_VAC_HYS := iq_stValve.rHYST_PERC * iq_stValve.rAT_VAC_SP;
END_IF

iq_stValve.rAT_VAC_HYS := LIMIT(0, iq_stValve.rAT_VAC_HYS, iq_stValve.rAT_VAC_SP);
IF iq_stValve.rAT_VAC_SP <> 0 THEN
	IF iq_stValve.rHYST_PERC <> (iq_stValve.rAT_VAC_HYS / iq_stValve.rAT_VAC_SP) THEN
		iq_stValve.rHYST_PERC := LIMIT(0, (iq_stValve.rAT_VAC_HYS / iq_stValve.rAT_VAC_SP) ,1);
	END_IF
END_IF
// Valve at vacuum check
///////////////////////////////////////////////////
	set := i_stUSG.rPRESS < iq_stValve.rAT_VAC_HYS AND i_stDSG.rPRESS < iq_stValve.rAT_VAC_HYS AND i_stUSG.xPRESS_OK AND i_stDSG.xPRESS_OK;
 	iq_stValve.xAT_VAC S= set;
	reset := i_stUSG.rPRESS > iq_stValve.rAT_VAC_SP OR i_stDSG.rPRESS > iq_stValve.rAT_VAC_SP OR NOT i_stUSG.xPRESS_OK OR NOT i_stDSG.xPRESS_OK;
	iq_stValve.xAT_VAC R= reset;
	
// Differential pressure check
///////////////////////////////////////////////////
	(* Calc the differential pressure across the valve *)
	rDiffPress := ABS(i_stUSG.rPRESS - i_stDSG.rPRESS);
	
	(* As long as the differential pressure is less than 30mbar, the valve is allowed to open *)
	IF rDiffPress <= rDiffPressAllowed AND i_stUSG.xPRESS_OK AND i_stDSG.xPRESS_OK THEN
		iq_stValve.xDP_OK := TRUE;
	ELSE
		iq_stValve.xDP_OK	:= FALSE;
		(* If the differential pressure is exceeded, even when the valve is open,
		the state is unexpected and triggers a fault, because it suggests that something
		is wrong with the valve, or gauges or mapping or there is a major leak on one side.*)
		iq_stValve.eVGC_State := ERR_DiffPress;
	END_IF

// Valve state
///////////////////////////////////////////////////
CASE iq_stValve.eVGC_State OF
	Vented: (* The Vented state is used during pump down *)
		(* Assuming the pump down went well, we are now at vacuum on both sides,
		so we move to the vacuum state, otherwise remain in the vented state *)
		IF iq_stValve.xAT_VAC THEN
		iq_stValve.eVGC_State := AtVacuum;
		ELSE
		iq_stValve.eVGC_State := Vented;
		END_IF
	
	AtVacuum:
		IF iq_stValve.xAT_VAC THEN
		(* If both pressure setpoints are made,
		then enable the differential pressure interlock, regardless of the valve state
		assuming we're using some kind of ion gauge where a pressure setpoint cannot be higher than 1E-4 T *)
		iq_stValve.eVGC_State := AtVacuum;
		ELSE
		
			(* If the valve is open (or in an unknown state) and either gauge is not at it's vacuum setpoint,
			we have a loss of vacuum error *)
			IF (iq_stValve.i_xOpnLS OR (NOT iq_stValve.i_xOpnLS AND NOT iq_stValve.i_xClsLS)) THEN
			iq_stValve.eVGC_State := ERR_LostVac;
		
			(* Alternatively, if the valve is already closed and we lose pressure on one side,
			it was probably intentional venting, so we calmly move back to venting mode, and
			disable the differential pressure interlock *) //?? 
			ELSIF iq_stValve.i_xClsLS THEN
			iq_stValve.eVGC_State := Vented;
			END_IF
		
		END_IF
	
	ERR_DiffPress:
		iq_stValve.eVGC_State := Vented;
		iq_stValve.xERR_DifPres := TRUE;
	
	ERR_LostVac:
		iq_stValve.eVGC_State := Vented;
		iq_stValve.xERR_LstVac := TRUE;
	
	END_CASE




// Interlock evaluation - with bypass for DP ILK bypass
///////////////////////////////////////////////
IF i_xDis_DPIlk THEN
	iq_stValve.xOPN_OK := iq_stValve.xEXT_OK; // AND iq_stValve.xDP_OK ;
ELSE
	iq_stValve.xOPN_OK := iq_stValve.xEXT_OK AND iq_stValve.xAT_VAC;
END_IF


(* Valve operation *)

(* Override logic *)
(* Goal: give ability to override, but do so in a way that people won't forget it.
Solution: Override only after ten seconds of override, protect against blips,
when the valve permission goes true for more than ten seconds consistently, remove override
*)

tonDelOK(IN:=iq_stValve.xOPN_OK, PT:=tDelOK);
rtOK(CLK:=tonDelOK.Q);
IF rtOK.Q AND iq_stValve.pv_xOvrdOpn THEN 
iq_stValve.pv_xOvrdOpn :=FALSE;
iq_stValve.pv_xOPN_SW := TRUE; //for seamless transition
END_IF

//Override timer
tonOvrd(IN:=iq_stValve.pv_xOvrdOpn, PT:=tOvrd);

(* If Epics Command is to close the Valve, check if MPS and EPS are ok, otherwive Keep command set to open valve *)
IF NOT(iq_stValve.pv_xOPN_SW) AND ((NOT i_xPMPS_OK) OR (NOT i_xEPS_OK)) THEN
	iq_stValve.pv_xOPN_SW := TRUE;
END_IF
(* Reset the EPICS command to open the valve if the interlock is lost *) 
(* based on EPS ok state, EPS overrides OPN_OK*)
IF NOT iq_stValve.xOPN_OK THEN
	IF i_xEPS_OK THEN iq_stValve.pv_xOPN_SW := FALSE;
	ELSE iq_stValve.pv_xOPN_SW := TRUE;		
	END_IF
END_IF

(* Here's where the valve opens *)
iq_stValve.q_xOPN_DO := (iq_stValve.pv_xOPN_SW AND iq_stValve.xOPN_OK) OR (tonOvrd.Q AND g_stSystem.xOverrideMode);

(* When the valve looses its open limit switch signal it should alert MPS*)
xMPS_FAULT := NOT iq_stValve.i_xOpnLS; 

///Check valve postion timout
IF NOT iq_stValve.i_xClsLS AND tCLStimeout.Q THEN 
	iq_stValve.bErrorPresent := TRUE;
ELSIF NOT iq_stValve.i_xOpnLS AND tOPNtimeout.Q THEN 
	iq_stValve.bErrorPresent := TRUE;
END_IF

(*Timers*)
tOPNtimeout(IN:= iq_stValve.q_xOPN_DO, PT := tTimeOutDuration );
tCLStimeout(IN:= NOT iq_stValve.q_xOPN_DO, PT := tTimeOutDuration);


// Alarm reset
//////////////////////////////////////
ACT_ResetAlarms();

(*IO Mapping*)
ACT_IO();

ACTION ACT_IO:
(*inputs*)
iq_stValve.i_xOpnLS := 	i_xOpnLS;
iq_stValve.i_xClsLS:=	i_xClsLS;
iq_stValve.xEXT_OK := i_xEXT_OK;
(*outputs*)
q_xOPN_DO:= iq_stValve.q_xOPN_DO;
END_ACTION

ACTION ACT_ResetAlarms:
iq_stValve.xERR_DifPres R= iq_stValve.pv_xAlmRst;
iq_stValve.xERR_LstVac R= iq_stValve.pv_xAlmRst;
iq_stValve.bErrorPresent R= iq_stValve.pv_xAlmRst;
END_ACTION

END_FUNCTION_BLOCK

// POUs/Functions/Valves/FB_VRC
FUNCTION_BLOCK FB_VRC
VAR_IN_OUT
	
END_VAR
VAR_INPUT
	
END_VAR
VAR_OUTPUT
	{attribute 'pytmc' := '
    pv:
	'}
	iq_stValve : ST_VRC;
END_VAR
VAR

tonOvrd	:	TON;
tonDelOK : TON;
rtOK	:	R_TRIG;


	(*IO*)
	i_xOpnLS	AT%I*: BOOL;
	i_xClsLS	AT%I*: BOOL;
	q_xOPN_DO	AT%Q*: BOOL;
END_VAR


///Check valve postion
IF NOT iq_stValve.i_xClsLS AND iq_stValve.i_xOpnLS THEN 
	iq_stValve.eState:=0;
ELSIF iq_stValve.i_xClsLS AND NOT iq_stValve.i_xOpnLS THEN 
	iq_stValve.eState:=1;
ELSIF NOT iq_stValve.i_xClsLS AND NOT iq_stValve.i_xOpnLS THEN 
	iq_stValve.eState:=2;
ELSE
	iq_stValve.eState:=3;
END_IF

IF NOT iq_stValve.xOPN_OK and NOT tonOvrd.Q THEN
iq_stValve.pv_xOPN_SW := FALSE;
END_IF

(* Override logic *)
(* Goal: give ability to override, but do so in a way that people won't forget it.
Solution: Override only after ten seconds of override, protect against blips,
when the valve permission goes true for more than ten seconds consistently, remove override
*)

tonDelOK(IN:=iq_stValve.xOPN_OK, PT:=T#10S);
rtOK(CLK:=tonDelOK.Q);
IF rtOK.Q THEN iq_stValve.pv_xOvrdOpn :=FALSE; END_IF

//Override timer
tonOvrd(IN:=iq_stValve.pv_xOvrdOpn, PT:=T#10S);

(* Here's where the valve opens *)
iq_stValve.q_xOPN_DO := (iq_stValve.pv_xOPN_SW AND iq_stValve.xOPN_OK) OR (tonOvrd.Q AND g_stSystem.xOverrideMode);

(*Soft IO Mapping*)
ACT_IO();

ACTION ACT_IO:
(*inputs*)
iq_stValve.i_xOpnLS := 	i_xOpnLS;
iq_stValve.i_xClsLS:=	i_xClsLS;
(*outputs*)
q_xOPN_DO:= iq_stValve.q_xOPN_DO;
END_ACTION

METHOD PUBLIC F_TURBO_VRC_ILK : BOOL
VAR_INPUT

	i_xHiVac 	: BOOL;
	i_xRunPTM	: BOOL;
	i_xFLVac	: BOOL;

END_VAR
VAR

	rHysterisis : REAL := 0;

	xInterlock: BOOL;
	rTolerance: REAL := 20;
END_VAR
(* Close the vic if the roughing pump pirani loses its at-vac setpoint while the turbo is pumping *)
F_TURBO_VRC_ILK := (NOT i_xHiVac AND NOT i_xRunPTM AND NOT i_xFLVac) OR
					(NOT i_xRunPTM AND i_xFLVac) OR
					(i_xRunPTM AND i_xFLVac);
END_METHOD

END_FUNCTION_BLOCK

// POUs/Functions/Valves/FB_VRC_OK_CLS
FUNCTION_BLOCK FB_VRC_OK_CLS
VAR_IN_OUT
	iq_stValve : ST_VRC;
END_VAR
VAR_INPUT

END_VAR
VAR_OUTPUT
END_VAR
VAR

tonOvrd	:	TON;
tonDelOK : TON;
rtOK	:	R_TRIG;

END_VAR

(* This fumction block is different from the regular VRC in that CLOSING must be permitted. *)
(* Implemented for the funky valve 04 on LAMP *)
IF NOT iq_stValve.xOPN_OK and NOT tonOvrd.Q THEN
iq_stValve.pv_xOPN_SW := FALSE;
END_IF

(* Override logic *)
(* Goal: give ability to override, but do so in a way that people won't forget it.
Solution: Override only after ten seconds of override, protect against blips,
when the valve permission goes true for more than ten seconds consistently, remove override
*)

tonDelOK(IN:=iq_stValve.xOPN_OK, PT:=T#10S);
rtOK(CLK:=tonDelOK.Q);
IF rtOK.Q THEN iq_stValve.pv_xOvrdOpn :=FALSE; END_IF

//Override timer
tonOvrd(IN:=iq_stValve.pv_xOvrdOpn, PT:=T#10S);

(* Here's where the valve opens *)
iq_stValve.q_xOPN_DO := NOT iq_stValve.xCLS_OK OR ((iq_stValve.pv_xOPN_SW AND iq_stValve.xOPN_OK) OR (tonOvrd.Q AND g_stSystem.xOverrideMode));

END_FUNCTION_BLOCK
